(* CODESYS project DCCM_PCL_2.project
   Author: jrfsc
   Version: 0.0.0.0
   Title: DCCM_PCL_2

Project tree, tasks and I/O mapping:
  DCCM_PCL_2 : TM251MESC, Schneider Electric, order no. TM251MESC, version 5.1.9.35
      settings: OPCUA enable = False
    application Application
      libraries: IecRtsServices, 1.0.4.0 (Schneider Electric)
      task MAST (cyclic, interval 20 ms, priority 15, watchdog 100 ms x 1) calls INPUT_MAPPING, ROOM_1, ROOM_2, ROOM_3, ROOM_4, OUTPUT_MAPPING, SR_Main
      global variables GVL
      program SR_Main [FBD]
      program INPUT_MAPPING [ST]
      program OUTPUT_MAPPING [ST]
      FBs/
        function block DUTY [ST]
        function block DUTY_CHANGE [ST]
        function block FB_9StatesMonitoring [ST]
        function block FB_DUTY_DUTY_STANDBY_PUMP_SPD [ST]
        function block FB_FLOATING_VALVE [ST]
        function block FB_HEATING_OR_COOLING [ST]
        function block FB_OMODE [ST]
        function block FB_PMODE [ST]
        function block FB_SETPOINT_MODE [ST]
        function block FB_WATCHDOG [ST]
        function block LINEAR [ST]
        function block SATSP_CALC [ST]
        function block SB_HEATING_COOLING [ST]
        function block TERMINAL_LOAD [ST]
        program ISO_MODE [ST]
      Enumeration/
        data type ET_9STATE_MONITORING
        data type ET_OMODE
        data type ET_PMODE
      LIBRARY/
        function block FB_PULSE_GENERATOR [ST]
        function block FB_0_10V_TO_2_10V_OUTPUT [ST]
        function block FB_PCMS_WATCHDOG [ST]
      Library/
        function block FB_SETPOINT_RAMPING [ST]
      program ROOM_1 [FBD]
      program ROOM_4 [FBD]
      program ROOM_3 [FBD]
      program ROOM_2 [FBD]
      global variables DCCMNVL
      program SendDeprox [CFC]
      global variables PersistentVars
    IO_Bus : IO bus - TM3, Schneider Electric, version 5.1.9.35
      Module_1 : TM3AQ4/G, Schneider Electric, order no. TM3AQ4/G, version 1.0.0.16
          settings: KPI Configuration.KPI Configuration = 16; KPI Configuration.KPI Configuration = 16; KPI Configuration.KPI Configuration = 16; KPI Configuration.KPI Configuration = 16; KPI Configuration.KPI Configuration = 0; KPI Configuration.KPI Configuration = 0; KPI Configuration.KPI Configuration = 0; KPI Configuration.KPI Configuration = 0; KPI Configuration.KPI Configuration = 16; KPI Configuration.KPI Configuration = 39; KPI Configuration.KPI Configuration = 16; KPI Configuration.KPI Configuration = 39; KPI Configuration.KPI Configuration = 16; KPI Configuration.KPI Configuration = 39; KPI Configuration.KPI Configuration = 16; KPI Configuration.KPI Configuration = 39
          output qRM1_TRANSFER_DAMPER : INT  // QW0
          output qRM2_TRANSFER_DAMPER : INT  // QW1
          output qRM3_TRANSFER_DAMPER : INT  // QW2
          output qRM4_TRANSFER_DAMPER : INT  // QW3
          input  ibModule_1_IBStatusQW0 : BYTE  // IBStatusQW0
          input  ibModule_1_IBStatusQW1 : BYTE  // IBStatusQW1
          input  ibModule_1_IBStatusQW2 : BYTE  // IBStatusQW2
          input  ibModule_1_IBStatusQW3 : BYTE  // IBStatusQW3
      Module_2 : TM3AI8/G, Schneider Electric, order no. TM3AI8/G, version 1.0.0.27
          settings: KPI Configuration.KPI Configuration = 32; KPI Configuration.KPI Configuration = 32; KPI Configuration.KPI Configuration = 32; KPI Configuration.KPI Configuration = 32; KPI Configuration.KPI Configuration = 32; KPI Configuration.KPI Configuration = 32; KPI Configuration.KPI Configuration = 32; KPI Configuration.KPI Configuration = 32; KPI Configuration.KPI Configuration = 231; KPI Configuration.KPI Configuration = 255; KPI Configuration.KPI Configuration = 231; KPI Configuration.KPI Configuration = 255; KPI Configuration.KPI Configuration = 231; KPI Configuration.KPI Configuration = 255; KPI Configuration.KPI Configuration = 231; KPI Configuration.KPI Configuration = 255; KPI Configuration.KPI Configuration = 231; KPI Configuration.KPI Configuration = 255; KPI Configuration.KPI Configuration = 231; KPI Configuration.KPI Configuration = 255; KPI Configuration.KPI Configuration = 231; KPI Configuration.KPI Configuration = 255; KPI Configuration.KPI Configuration = 231; KPI Configuration.KPI Configuration = 255; KPI Configuration.KPI Configuration = 25; KPI Configuration.KPI Configuration = 0; KPI Configuration.KPI Configuration = 25; KPI Configuration.KPI Configuration = 0; KPI Configuration.KPI Configuration = 25; KPI Configuration.KPI Configuration = 0; KPI Configuration.KPI Configuration = 25; KPI Configuration.KPI Configuration = 0; KPI Configuration.KPI Configuration = 25; KPI Configuration.KPI Configuration = 0; KPI Configuration.KPI Configuration = 25; KPI Configuration.KPI Configuration = 0; KPI Configuration.KPI Configuration = 25; KPI Configuration.KPI Configuration = 0; KPI Configuration.KPI Configuration = 25; KPI Configuration.KPI Configuration = 0
          input  iRM1_DP_H_TO_R : INT  // IW0
          input  iRM1_DP_H_TO_A : INT  // IW1
          input  iRM1_DP_A_TO_R : INT  // IW2
          input  iRM2_DP_H_TO_R : INT  // IW3
          input  iRM2_DP_A_TO_R : INT  // IW4
          input  iRM2_3_DP_H_TO_A : INT  // IW5
          input  iRM3_DP_H_TO_R : INT  // IW6
          input  iRM3_DP_A_TO_R : INT  // IW7
          input  ibModule_2_IBStatusIW0 : BYTE  // IBStatusIW0
          input  ibModule_2_IBStatusIW1 : BYTE  // IBStatusIW1
          input  ibModule_2_IBStatusIW2 : BYTE  // IBStatusIW2
          input  ibModule_2_IBStatusIW3 : BYTE  // IBStatusIW3
          input  ibModule_2_IBStatusIW4 : BYTE  // IBStatusIW4
          input  ibModule_2_IBStatusIW5 : BYTE  // IBStatusIW5
          input  ibModule_2_IBStatusIW6 : BYTE  // IBStatusIW6
          input  ibModule_2_IBStatusIW7 : BYTE  // IBStatusIW7
      Module_3 : TM3AM6/G, Schneider Electric, order no. TM3AM6/G, version 1.0.0.23
          settings: KPI Configuration.KPI Configuration = 32; KPI Configuration.KPI Configuration = 32; KPI Configuration.KPI Configuration = 32; KPI Configuration.KPI Configuration = 32; KPI Configuration.KPI Configuration = 231; KPI Configuration.KPI Configuration = 255; KPI Configuration.KPI Configuration = 231; KPI Configuration.KPI Configuration = 255; KPI Configuration.KPI Configuration = 231; KPI Configuration.KPI Configuration = 255; KPI Configuration.KPI Configuration = 0; KPI Configuration.KPI Configuration = 25; KPI Configuration.KPI Configuration = 0; KPI Configuration.KPI Configuration = 25; KPI Configuration.KPI Configuration = 0; KPI Configuration.KPI Configuration = 25; KPI Configuration.KPI Configuration = 0; KPI Configuration.KPI Configuration = 100; KPI Configuration.KPI Configuration = 0
          input  iRM4_DP_H_TO_R : INT  // IW0
          input  iRM4_DP_H_TO_A : INT  // IW1
          input  iRM4_DP_A_TO_R : INT  // IW2
          input  iRM1_TRANSFER_DAMPER_FB : INT  // IW3
          input  ibModule_3_IBStatusIW0 : BYTE  // IBStatusIW0
          input  ibModule_3_IBStatusIW1 : BYTE  // IBStatusIW1
          input  ibModule_3_IBStatusIW2 : BYTE  // IBStatusIW2
          input  ibModule_3_IBStatusIW3 : BYTE  // IBStatusIW3
          input  ibModule_3_IBStatusQW0 : BYTE  // IBStatusQW0
          input  ibModule_3_IBStatusQW1 : BYTE  // IBStatusQW1
          unmapped channels: QW0, QW1
      Module_4 : TM3AM6/G, Schneider Electric, order no. TM3AM6/G, version 1.0.0.23
          settings: KPI Configuration.KPI Configuration = 32; KPI Configuration.KPI Configuration = 32; KPI Configuration.KPI Configuration = 32; KPI Configuration.KPI Configuration = 0; KPI Configuration.KPI Configuration = 0; KPI Configuration.KPI Configuration = 0; KPI Configuration.KPI Configuration = 100; KPI Configuration.KPI Configuration = 0; KPI Configuration.KPI Configuration = 100; KPI Configuration.KPI Configuration = 0; KPI Configuration.KPI Configuration = 100; KPI Configuration.KPI Configuration = 0
          input  iRM2_TRANSFER_DAMPER_FB : INT  // IW0
          input  iRM3_TRANSFER_DAMPER_FB : INT  // IW1
          input  iRM4_TRANSFER_DAMPER_FB : INT  // IW2
          input  ibModule_4_IBStatusIW0 : BYTE  // IBStatusIW0
          input  ibModule_4_IBStatusIW1 : BYTE  // IBStatusIW1
          input  ibModule_4_IBStatusIW2 : BYTE  // IBStatusIW2
          input  ibModule_4_IBStatusIW3 : BYTE  // IBStatusIW3
          input  ibModule_4_IBStatusQW0 : BYTE  // IBStatusQW0
          input  ibModule_4_IBStatusQW1 : BYTE  // IBStatusQW1
          unmapped channels: IW3, QW0, QW1
      Module_5 : TM3DM24R/G, Schneider Electric, order no. TM3DM24R/G, version 1.0.2.0
          input  iRM1_SUPPLY_DAMPER_STS : BOOL  // IW0.I0
          input  iRM2_SUPPLY_DAMPER_STS : BOOL  // IW0.I1
          input  iRM3_SUPPLY_DAMPER_STS : BOOL  // IW0.I2
          input  iRM4_SUPPLY_DAMPER_STS : BOOL  // IW0.I3
          input  iRM1_EXHAUST_DAMPER_STS : BOOL  // IW0.I4
          input  iRM2_EXHAUST_DAMPER_STS : BOOL  // IW0.I5
          input  iRM3_EXHAUST_DAMPER_STS : BOOL  // IW0.I6
          input  iRM4_EXHAUST_DAMPER_STS : BOOL  // IW0.I7
          input  iRM1_ISOLATION_MODE_SW : BOOL  // IW0.I8
          input  iRM1_DEPROX_MODE_SW : BOOL  // IW0.I9
          input  iRM1_ALARM_MUTE : BOOL  // IW0.I10
          input  iRM2_ISOLATION_MODE_SW : BOOL  // IW0.I11
          input  iRM2_DEPROX_MODE_SW : BOOL  // IW0.I12
          input  iRM2_ALARM_MUTE : BOOL  // IW0.I13
          input  iRM3_ISOLATION_MODE_SW : BOOL  // IW0.I14
          input  iRM3_DEPROX_MODE_SW : BOOL  // IW0.I15
          output qRM1_SUPPLY_DAMPER : BOOL  // QB0.Q0
          output qRM2_SUPPLY_DAMPER : BOOL  // QB0.Q1
          output qRM3_SUPPLY_DAMPER : BOOL  // QB0.Q2
          output qRM4_SUPPLY_DAMPER : BOOL  // QB0.Q3
          output qRM1_EXHAUST_DAMPER : BOOL  // QB0.Q4
          output qRM2_EXHAUST_DAMPER : BOOL  // QB0.Q5
          output qRM3_EXHAUST_DAMPER : BOOL  // QB0.Q6
          output qRM4_EXHAUST_DAMPER : BOOL  // QB0.Q7
          unmapped channels: IW0, QB0
      Module_6 : TM3DM24R/G, Schneider Electric, order no. TM3DM24R/G, version 1.0.2.0
          input  iRM3_ALARM_MUTE : BOOL  // IW0.I0
          input  iRM4_ISOLATION_MODE_SW : BOOL  // IW0.I1
          input  iRM4_DEPROX_MODE_SW : BOOL  // IW0.I2
          input  iRM4_ALARM_MUTE : BOOL  // IW0.I3
          output qRM1_NEGATIVE_LED : BOOL  // QB0.Q0
          output qRM1_DEPROX_LED : BOOL  // QB0.Q1
          output qRM1_ALARM_LED : BOOL  // QB0.Q2
          output qRM1_STANDBY_LED : BOOL  // QB0.Q3
          output qRM2_NEGATIVE_LED : BOOL  // QB0.Q4
          output qRM2_DEPROX_LED : BOOL  // QB0.Q5
          output qRM2_ALARM_LED : BOOL  // QB0.Q6
          output qRM2_STANDBY_LED : BOOL  // QB0.Q7
          unmapped channels: IW0, QB0
      Module_7 : TM3DQ16R/G, Schneider Electric, order no. TM3DQ16R/G, version 1.0.1.14
          output qRM3_NEGATIVE_LED : BOOL  // QW0.Q0
          output qRM3_DEPROX_LED : BOOL  // QW0.Q1
          output qRM3_ALARM_LED : BOOL  // QW0.Q2
          output qRM3_STANDBY_LED : BOOL  // QW0.Q3
          output qRM4_NEGATIVE_LED : BOOL  // QW0.Q4
          output qRM4_DEPROX_LED : BOOL  // QW0.Q5
          output qRM4_ALARM_LED : BOOL  // QW0.Q6
          output qRM4_STANDBY_LED : BOOL  // QW0.Q7
          output qRM1_BUZZER : BOOL  // QW0.Q8
          output qRM2_BUZZER : BOOL  // QW0.Q9
          output qRM3_BUZZER : BOOL  // QW0.Q10
          output qRM4_BUZZER : BOOL  // QW0.Q11
          unmapped channels: QW0
    COM_Bus : COM bus, Schneider Electric, version 5.1.9.35
    Ethernet_1 : Ethernet Network, Schneider Electric, version 5.1.9.35
        settings: WebServer = TRUE; FTP Server = FALSE; SoMachine Protocol = TRUE; Modbus Server = TRUE; NetManage Protocol = TRUE; SNMP protocol = FALSE; WebVisu protocol = FALSE; Secured Web Server = TRUE
    Serial_Line_1 : Serial line, Schneider Electric, version 5.1.9.35
      Machine_Expert_Network_Manager : Machine Expert-Network Manager, Schneider Electric, version 4.0.0.4
    CAN_1 : CANopen bus, Schneider Electric, version 5.1.9.35
*)

// DCCM_PCL_2/Application/Enumeration/ET_9STATE_MONITORING
{attribute 'qualified_only' := ''}
{attribute 'strict' := ''}
TYPE ET_9STATE_MONITORING :
(
	STOPPED := 0,
	RUNNING := 1,
	STARTING := 2,
	STOPPING := 3,
	START_FAIL := 4,
	STOP_FAIL := 5,
	UNEXPECTED_START := 6,
	UNEXPECTED_STOP := 7,
	FIRE_STOP := 8,
	UNKNOWN := 9
);
END_TYPE

// DCCM_PCL_2/Application/Enumeration/ET_OMODE
{attribute 'qualified_only' := ''}
{attribute 'strict' := ''}
TYPE ET_OMODE :
(
	UNOCC := 0,
	OPTSTART := 1,
	SCH := 2,
	AHRS := 3,
	MOTDETECT := 4,
	SETBACK := 7
);
END_TYPE

// DCCM_PCL_2/Application/Enumeration/ET_PMODE
{attribute 'qualified_only' := ''}
{attribute 'strict' := ''}
TYPE ET_PMODE :
(
	OFF_NORMAL := 0,
	OFF_PCMS := 1,
	OFF_Fire := 2,
	OFF_DMPRLOCK := 3,
	OFF_RESET := 4,
	Startup := 5,
	Purge := 6,
	RUN_NORMAL := 7
);
END_TYPE

// DCCM_PCL_2/Application/GVL
{attribute 'qualified_only'}
VAR_GLOBAL
	RM1_TRANSFER_DAMPER AT %MD500: REAL;
	RM2_TRANSFER_DAMPER AT %MD501: REAL;
	RM3_TRANSFER_DAMPER AT %MD502: REAL;
	RM4_TRANSFER_DAMPER AT %MD503: REAL;
	RM1_DP_H_TO_R AT %MD504: REAL;
	RM1_DP_H_TO_A AT %MD505: REAL;
	RM1_DP_A_TO_R AT %MD506: REAL;
	RM2_DP_H_TO_R AT %MD507: REAL;
	RM2_DP_A_TO_R AT %MD508: REAL;
	RM2_3_DP_H_TO_A AT %MD509: REAL;
	RM3_DP_H_TO_R AT %MD510: REAL;
	RM3_DP_A_TO_R AT %MD511: REAL;
	RM4_DP_H_TO_R AT %MD512: REAL;
	RM4_DP_H_TO_A AT %MD513: REAL;
	RM4_DP_A_TO_R AT %MD514: REAL;
	RM1_TRANSFER_DAMPER_FB AT %MD515: REAL;
	RM2_TRANSFER_DAMPER_FB AT %MD516: REAL;
	RM3_TRANSFER_DAMPER_FB AT %MD517: REAL;
	RM4_TRANSFER_DAMPER_FB AT %MD518: REAL;
	RM1_SUPPLY_DAMPER_STS AT %MX0.0: BOOL;
	RM2_SUPPLY_DAMPER_STS AT %MX0.1: BOOL;
	RM3_SUPPLY_DAMPER_STS AT %MX0.2: BOOL;
	RM4_SUPPLY_DAMPER_STS AT %MX0.3: BOOL;
	RM1_EXHAUST_DAMPER_STS AT %MX0.4: BOOL;
	RM2_EXHAUST_DAMPER_STS AT %MX0.5: BOOL;
	RM3_EXHAUST_DAMPER_STS AT %MX0.6: BOOL;
	RM4_EXHAUST_DAMPER_STS AT %MX0.7: BOOL;
	RM1_ISOLATION_MODE_SW AT %MX1.0: BOOL;
	RM1_DEPROX_MODE_SW AT %MX1.1: BOOL;
	RM1_ALARM_MUTE_SW AT %MX1.2: BOOL;
	RM2_ISOLATION_MODE_SW AT %MX1.3: BOOL;
	RM2_DEPROX_MODE_SW AT %MX1.4: BOOL;
	RM2_ALARM_MUTE_SW AT %MX1.5: BOOL;
	RM3_ISOLATION_MODE_SW AT %MX1.6: BOOL;
	RM3_DEPROX_MODE_SW AT %MX1.7: BOOL;
	RM1_SUPPLY_DAMPER AT %MX2.0: BOOL;
	RM2_SUPPLY_DAMPER AT %MX2.1: BOOL;
	RM3_SUPPLY_DAMPER AT %MX2.2: BOOL;
	RM4_SUPPLY_DAMPER AT %MX2.3: BOOL;
	RM1_EXHAUST_DAMPER AT %MX2.4: BOOL;
	RM2_EXHAUST_DAMPER AT %MX2.5: BOOL;
	RM3_EXHAUST_DAMPER AT %MX2.6: BOOL;
	RM4_EXHAUST_DAMPER AT %MX2.7: BOOL;
	RM3_ALARM_MUTE AT %MX3.0: BOOL;
	RM4_ISOLATION_MODE_SW AT %MX3.1: BOOL;
	RM4_DEPROX_MODE_SW AT %MX3.2: BOOL;
	RM4_ALARM_MUTE AT %MX3.3: BOOL;
	RM1_NEGATIVE_LED AT %MX3.4: BOOL;
	RM1_DEPROX_LED AT %MX3.5: BOOL;
	RM1_ALARM_LED AT %MX3.6: BOOL;
	RM1_STANDBY_LED AT %MX3.7: BOOL;
	RM2_NEGATIVE_LED AT %MX4.0: BOOL;
	RM2_DEPROX_LED AT %MX4.1: BOOL;
	RM2_ALARM_LED AT %MX4.2: BOOL;
	RM2_STANDBY_LED AT %MX4.3: BOOL;
	RM3_NEGATIVE_LED AT %MX4.4: BOOL;
	RM3_DEPROX_LED AT %MX4.5: BOOL;
	RM3_ALARM_LED AT %MX4.6: BOOL;
	RM3_STANDBY_LED AT %MX4.7: BOOL;
	RM4_NEGATIVE_LED AT %MX5.0: BOOL;
	RM4_ALARM_LED AT %MX5.1: BOOL;
	RM4_STANDBY_LED AT %MX5.2: BOOL;
	RM4_DEPROX_LED AT %MX5.3: BOOL;
	RM1_BUZZER AT %MX5.4: BOOL;
	RM2_BUZZER AT %MX5.5: BOOL;
	RM3_BUZZER AT %MX5.6: BOOL;
	RM4_BUZZER AT %MX5.7: BOOL;
	RM1_ISO_MODE AT %MW9000: INT;
	RM2_ISO_MODE AT %MW9001: INT;
	RM3_ISO_MODE AT %MW9002: INT;
	RM4_ISO_MODE AT %MW9003: INT;
	RM1_TRANSFER_DAMPER_MAN AT %MD523: REAL;
END_VAR
VAR_GLOBAL RETAIN PERSISTENT
	RM1_TRANSFER_DAMPER_MD AT %MX6.0: BOOL := TRUE;
END_VAR
VAR_GLOBAL
	RM2_TRANSFER_DAMPER_MAN AT %MD524: REAL;
END_VAR
VAR_GLOBAL RETAIN PERSISTENT
	RM2_TRANSFER_DAMPER_MD AT %MX6.1: BOOL := TRUE;
END_VAR
VAR_GLOBAL
	RM3_TRANSFER_DAMPER_MAN AT %MD525: REAL;
END_VAR
VAR_GLOBAL RETAIN PERSISTENT
	RM3_TRANSFER_DAMPER_MD AT %MX6.2: BOOL := TRUE;
END_VAR
VAR_GLOBAL
	RM4_TRANSFER_DAMPER_MAN AT %MD526: REAL;
END_VAR
VAR_GLOBAL RETAIN PERSISTENT
	RM4_TRANSFER_DAMPER_MD AT %MX6.3: BOOL := TRUE;
	RM1_DP1_SP AT %MD527: REAL := 8;
	RM2_DP1_SP AT %MD528: REAL := 8;
	RM3_DP1_SP AT %MD529: REAL := 8;
	RM4_DP1_SP AT %MD530: REAL := 8;
END_VAR
VAR_GLOBAL
	RM1_DP_ALM AT %MX6.4: BOOL;
	RM2_DP_ALM AT %MX6.5: BOOL;
	RM3_DP_ALM AT %MX6.6: BOOL;
	RM4_DP_ALM AT %MX6.7: BOOL;
	RM1_SUPPLY_DAMPER_MAN AT %MX7.0: BOOL;
END_VAR
VAR_GLOBAL RETAIN PERSISTENT
	RM1_SUPPLY_DAMPER_MD AT %MX7.1: BOOL := TRUE;
END_VAR
VAR_GLOBAL
	RM1_EXHAUST_DAMPER_MAN AT %MX7.2: BOOL;
END_VAR
VAR_GLOBAL RETAIN PERSISTENT
	RM1_EXHAUST_DAMPER_MD AT %MX7.3: BOOL := TRUE;
END_VAR
VAR_GLOBAL
	RM2_SUPPLY_DAMPER_MAN AT %MX7.4: BOOL;
END_VAR
VAR_GLOBAL RETAIN PERSISTENT
	RM2_SUPPLY_DAMPER_MD AT %MX7.5: BOOL := TRUE;
END_VAR
VAR_GLOBAL
	RM2_EXHAUST_DAMPER_MAN AT %MX7.6: BOOL;
END_VAR
VAR_GLOBAL RETAIN PERSISTENT
	RM2_EXHAUST_DAMPER_MD AT %MX7.7: BOOL := TRUE;
END_VAR
VAR_GLOBAL
	RM3_SUPPLY_DAMPER_MAN AT %MX8.0: BOOL;
END_VAR
VAR_GLOBAL RETAIN PERSISTENT
	RM3_SUPPLY_DAMPER_MD AT %MX8.1: BOOL := TRUE;
END_VAR
VAR_GLOBAL
	RM3_EXHAUST_DAMPER_MAN AT %MX8.2: BOOL;
END_VAR
VAR_GLOBAL RETAIN PERSISTENT
	RM3_EXHAUST_DAMPER_MD AT %MX8.3: BOOL := TRUE;
END_VAR
VAR_GLOBAL
	RM4_SUPPLY_DAMPER_MAN AT %MX8.4: BOOL;
END_VAR
VAR_GLOBAL RETAIN PERSISTENT
	RM4_SUPPLY_DAMPER_MD AT %MX8.5: BOOL := TRUE;
END_VAR
VAR_GLOBAL
	RM4_EXHAUST_DAMPER_MAN AT %MX8.6: BOOL;
END_VAR
VAR_GLOBAL RETAIN PERSISTENT
	RM4_EXHAUST_DAMPER_MD AT %MX8.7: BOOL := TRUE;
END_VAR
VAR_GLOBAL
	RM1_NEGATIVE_LED_MAN: BOOL;
	RM1_NEGATIVE_LED_MD: BOOL := TRUE;
	RM1_DEPROX_LED_MAN: BOOL;
	RM1_DEPROX_LED_MD: BOOL := TRUE;
	RM1_ALARM_LED_MAN: BOOL;
	RM1_ALARM_LED_MD: BOOL := TRUE;
	RM1_STANDBY_LED_MAN: BOOL;
	RM1_STANDBY_LED_MD: BOOL := TRUE;
	RM2_NEGATIVE_LED_MAN: BOOL;
	RM2_NEGATIVE_LED_MD: BOOL := TRUE;
	RM2_DEPROX_LED_MAN: BOOL;
	RM2_DEPROX_LED_MD: BOOL := TRUE;
	RM2_STANDBY_LED_MAN: BOOL;
	RM2_STANDBY_LED_MD: BOOL := TRUE;
	RM2_ALARM_LED_MAN: BOOL;
	RM2_ALARM_LED_MD: BOOL := TRUE;
	RM3_NEGATIVE_LED_MAN: BOOL;
	RM3_NEGATIVE_LED_MD: BOOL := TRUE;
	RM3_DEPROX_LED_MAN: BOOL;
	RM3_DEPROX_LED_MD: BOOL := TRUE;
	RM3_ALARM_LED_MAN: BOOL;
	RM3_ALARM_LED_MD: BOOL := TRUE;
	RM3_STANDBY_LED_MAN: BOOL;
	RM3_STANDBY_LED_MD: BOOL := TRUE;
	RM4_NEGATIVE_LED_MAN: BOOL;
	RM4_NEGATIVE_LED_MD: BOOL := TRUE;
	RM4_DEPROX_LED_MAN: BOOL;
	RM4_DEPROX_LED_MD: BOOL := TRUE;
	RM4_ALARM_LED_MAN: BOOL;
	RM4_ALARM_LED_MD: BOOL := TRUE;
	RM4_STANDBY_LED_MAN: BOOL;
	RM4_STANDBY_LED_MD: BOOL := TRUE;
END_VAR
VAR_GLOBAL RETAIN PERSISTENT
	RM1_TRANSFER_DAMPER_ISO_SP AT %MD535: REAL := 15;
	RM2_TRANSFER_DAMPER_ISO_SP AT %MD536: REAL := 15;
	RM3_TRANSFER_DAMPER_ISO_SP AT %MD537: REAL := 15;
	RM4_TRANSFER_DAMPER_ISO_SP AT %MD538: REAL := 10;
END_VAR
VAR_GLOBAL
	RM1_BUZZER_MAN: BOOL;
	RM1_BUZZER_MD: BOOL := TRUE;
	RM2_BUZZER_MAN: BOOL;
	RM2_BUZZER_MD: BOOL := TRUE;
	RM3_BUZZER_MAN: BOOL;
	RM3_BUZZER_MD: BOOL := TRUE;
	RM4_BUZZER_MAN: BOOL;
	RM4_BUZZER_MD: BOOL := TRUE;
END_VAR
VAR_GLOBAL RETAIN PERSISTENT
	RM1_ALARM_DELAY AT %MD539: real := 180;
	RM2_ALARM_DELAY AT %MD540: real := 180;
	RM3_ALARM_DELAY AT %MD541: real := 180;
	RM4_ALARM_DELAY AT %MD542: real := 180;
END_VAR
VAR_GLOBAL
	DEPROX_TOTAL AT %MW9004: INT;
END_VAR
VAR_GLOBAL RETAIN PERSISTENT
	RM1_DP2_SP AT %MD543: REAL;
	RM1_DP3_SP AT %MD544: REAL;
	RM2_DP2_SP AT %MD545: REAL;
	RM2_DP3_SP AT %MD546: REAL;
	RM3_DP2_SP AT %MD547: REAL;
	RM3_DP3_SP AT %MD548: REAL;
	RM4_DP2_SP AT %MD549: REAL;
	RM4_DP3_SP AT %MD550: REAL;
	RM1_TRANSFER_DAMPER_DEP_SP AT %MD551: REAL;
	RM2_TRANSFER_DAMPER_DEP_SP AT %MD552: REAL;
	RM3_TRANSFER_DAMPER_DEP_SP AT %MD553: REAL;
	RM4_TRANSFER_DAMPER_DEP_SP AT %MD554: REAL;
END_VAR

// DCCM_PCL_2/Application/DCCMNVL
{attribute 'qualified_only'}
VAR_GLOBAL
	RM1_ISO_MODE AT %MW9000: INT;
	RM2_ISO_MODE AT %MW9001: INT;
	RM3_ISO_MODE AT %MW9002: INT;
	RM4_ISO_MODE AT %MW9003: INT;
END_VAR

// DCCM_PCL_2/Application/PersistentVars
{attribute 'qualified_only'}
VAR_GLOBAL PERSISTENT RETAIN
	// Generated instance path of persistent variable
	GVL.RM1_TRANSFER_DAMPER_MD: BOOL := TRUE;
	// Generated instance path of persistent variable
	GVL.RM2_TRANSFER_DAMPER_MD: BOOL := TRUE;
	// Generated instance path of persistent variable
	GVL.RM3_TRANSFER_DAMPER_MD: BOOL := TRUE;
	// Generated instance path of persistent variable
	GVL.RM4_TRANSFER_DAMPER_MD: BOOL := TRUE;
	// Generated instance path of persistent variable
	GVL.RM1_DP1_SP: REAL := -5;
	// Generated instance path of persistent variable
	GVL.RM2_DP1_SP: REAL := -5;
	// Generated instance path of persistent variable
	GVL.RM3_DP1_SP: REAL := -5;
	// Generated instance path of persistent variable
	GVL.RM4_DP1_SP: REAL := -5;
	// Generated instance path of persistent variable
	GVL.RM1_SUPPLY_DAMPER_MD: BOOL := TRUE;
	// Generated instance path of persistent variable
	GVL.RM1_EXHAUST_DAMPER_MD: BOOL := TRUE;
	// Generated instance path of persistent variable
	GVL.RM2_SUPPLY_DAMPER_MD: BOOL := TRUE;
	// Generated instance path of persistent variable
	GVL.RM2_EXHAUST_DAMPER_MD: BOOL := TRUE;
	// Generated instance path of persistent variable
	GVL.RM3_SUPPLY_DAMPER_MD: BOOL := TRUE;
	// Generated instance path of persistent variable
	GVL.RM3_EXHAUST_DAMPER_MD: BOOL := TRUE;
	// Generated instance path of persistent variable
	GVL.RM4_SUPPLY_DAMPER_MD: BOOL := TRUE;
	// Generated instance path of persistent variable
	GVL.RM4_EXHAUST_DAMPER_MD: BOOL := TRUE;
	// Generated instance path of persistent variable
	GVL.RM1_TRANSFER_DAMPER_ISO_SP: REAL := 15.0;
	// Generated instance path of persistent variable
	GVL.RM2_TRANSFER_DAMPER_ISO_SP: REAL := 15.0;
	// Generated instance path of persistent variable
	GVL.RM3_TRANSFER_DAMPER_ISO_SP: REAL := 15.0;
	// Generated instance path of persistent variable
	GVL.RM4_TRANSFER_DAMPER_ISO_SP: REAL := 10.0;
	// Generated instance path of persistent variable
	GVL.RM1_ALARM_DELAY: REAL := 180.0;
	// Generated instance path of persistent variable
	GVL.RM2_ALARM_DELAY: REAL := 180.0;
	// Generated instance path of persistent variable
	GVL.RM3_ALARM_DELAY: REAL := 180.0;
	// Generated instance path of persistent variable
	GVL.RM4_ALARM_DELAY: REAL := 180.0;
	// Generated instance path of persistent variable
	GVL.RM1_DP2_SP: REAL := -5;
	// Generated instance path of persistent variable
	GVL.RM1_DP3_SP: REAL := -5;
	// Generated instance path of persistent variable
	GVL.RM2_DP2_SP: REAL := -5;
	// Generated instance path of persistent variable
	GVL.RM2_DP3_SP: REAL := -5;
	// Generated instance path of persistent variable
	GVL.RM3_DP2_SP: REAL := -5;
	// Generated instance path of persistent variable
	GVL.RM3_DP3_SP: REAL := -5;
	// Generated instance path of persistent variable
	GVL.RM4_DP2_SP: REAL := -5;
	// Generated instance path of persistent variable
	GVL.RM4_DP3_SP: REAL := -5;
	// Generated instance path of persistent variable
	GVL.RM1_TRANSFER_DAMPER_DEP_SP: REAL;
	// Generated instance path of persistent variable
	GVL.RM2_TRANSFER_DAMPER_DEP_SP: REAL;
	// Generated instance path of persistent variable
	GVL.RM3_TRANSFER_DAMPER_DEP_SP: REAL;
	// Generated instance path of persistent variable
	GVL.RM4_TRANSFER_DAMPER_DEP_SP: REAL;
END_VAR

// DCCM_PCL_2/Application/INPUT_MAPPING
PROGRAM INPUT_MAPPING
VAR
		voltage_converter: FB_0_10V_TO_2_10V_OUTPUT;
END_VAR

//MAPPING HARDWARE INPUTS TO MEMORY WORDS

GVL.RM1_DP_H_TO_R := TO_REAL(iRM1_DP_H_TO_R);								//MODULE 2 TM3AI8 INPUT 0
GVL.RM1_DP_H_TO_A := TO_REAL(iRM1_DP_H_TO_A);								//MODULE 2 TM3AI8 INPUT 1
GVL.RM1_DP_A_TO_R := TO_REAL(iRM1_DP_A_TO_R);								//MODULE 2 TM3AI8 INPUT 2
GVL.RM2_DP_H_TO_R := TO_REAL(IRM2_DP_H_TO_R);								//MODULE 2 TM3AI8 INPUT 3
GVL.RM2_DP_A_TO_R := TO_REAL(iRM2_DP_A_TO_R);								//MODULE 2 TM3AI8 INPUT 4
GVL.RM2_3_DP_H_TO_A := TO_REAL(iRM2_3_DP_H_TO_A);							//MODULE 2 TM3AI8 INPUT 5
GVL.RM3_DP_H_TO_R := TO_REAL(iRM3_DP_H_TO_R);								//MODULE 2 TM3AI8 INPUT 6
GVL.RM3_DP_A_TO_R := TO_REAL(iRM3_DP_A_TO_R);								//MODULE 2 TM3AI8 INPUT 7

GVL.RM4_DP_H_TO_R := TO_REAL(iRM4_DP_H_TO_R);								//MODULE 3 TM3AM6 INPUT 0
GVL.RM4_DP_H_TO_A := TO_REAL(iRM4_DP_H_TO_A);								//MODULE 3 TM3AM6 INPUT 1
GVL.RM4_DP_A_TO_R := TO_REAL(iRM4_DP_A_TO_R);		
						//MODULE 3 TM3AM6 INPUT 2
//GVL.RM1_TRANSFER_DAMPER_FB := TO_REAL(iRM1_TRANSFER_DAMPER_FB);				//MODULE 3 TM3AM6 INPUT 3
//GVL.RM2_TRANSFER_DAMPER_FB := TO_REAL(iRM2_TRANSFER_DAMPER_FB);				//MODULE 4 TM3AM6 INPUT 0
//GVL.RM3_TRANSFER_DAMPER_FB := TO_REAL(iRM3_TRANSFER_DAMPER_FB);				//MODULE 4 TM3AM6 INPUT 1
//GVL.RM4_TRANSFER_DAMPER_FB := TO_REAL(iRM4_TRANSFER_DAMPER_FB);				//MODULE 4 TM3AM6 INPUT 2


GVL.RM1_TRANSFER_DAMPER_FB :=100-((((iRM1_TRANSFER_DAMPER_FB-100) * 100/80))+100);
GVL.RM2_TRANSFER_DAMPER_FB :=100-((((iRM2_TRANSFER_DAMPER_FB-100) * 100/80))+100);
GVL.RM3_TRANSFER_DAMPER_FB :=100-((((iRM3_TRANSFER_DAMPER_FB-100) * 100/80))+100);
GVL.RM4_TRANSFER_DAMPER_FB :=100-((((iRM4_TRANSFER_DAMPER_FB-100) * 100/80))+100);  //AI0  0v=open 10v=close



GVL.RM1_SUPPLY_DAMPER_STS := iRM1_SUPPLY_DAMPER_STS;						//MODULE 5 TM3DM24R INPUT 0
GVL.RM2_SUPPLY_DAMPER_STS := iRM2_SUPPLY_DAMPER_STS;						//MODULE 5 TM3DM24R INPUT 1
GVL.RM3_SUPPLY_DAMPER_STS := iRM3_SUPPLY_DAMPER_STS;						//MODULE 5 TM3DM24R INPUT 2
GVL.RM4_SUPPLY_DAMPER_STS := iRM4_SUPPLY_DAMPER_STS;						//MODULE 5 TM3DM24R INPUT 3
GVL.RM1_EXHAUST_DAMPER_STS := iRM1_EXHAUST_DAMPER_STS;						//MODULE 5 TM3DM24R INPUT 4
GVL.RM2_EXHAUST_DAMPER_STS := iRM2_EXHAUST_DAMPER_STS;						//MODULE 5 TM3DM24R INPUT 5
GVL.RM3_EXHAUST_DAMPER_STS := iRM3_EXHAUST_DAMPER_STS;						//MODULE 5 TM3DM24R INPUT 6
GVL.RM4_EXHAUST_DAMPER_STS := iRM4_EXHAUST_DAMPER_STS;						//MODULE 5 TM3DM24R INPUT 7
GVL.RM1_ISOLATION_MODE_SW := iRM1_ISOLATION_MODE_SW;						//MODULE 5 TM3DM24R INPUT 8
GVL.RM1_DEPROX_MODE_SW := iRM1_DEPROX_MODE_SW;								//MODULE 5 TM3DM24R INPUT 9
GVL.RM1_ALARM_MUTE_SW := iRM1_ALARM_MUTE;									//MODULE 5 TM3DM24R INPUT 10
GVL.RM2_ISOLATION_MODE_SW := iRM2_ISOLATION_MODE_SW;						//MODULE 5 TM3DM24R INPUT 11
GVL.RM2_DEPROX_MODE_SW := iRM2_DEPROX_MODE_SW;								//MODULE 5 TM3DM24R INPUT 12
GVL.RM2_ALARM_MUTE_SW := iRM2_ALARM_MUTE;									//MODULE 5 TM3DM24R INPUT 13
GVL.RM3_ISOLATION_MODE_SW := iRM3_ISOLATION_MODE_SW;						//MODULE 5 TM3DM24R INPUT 14
GVL.RM3_DEPROX_MODE_SW := iRM3_DEPROX_MODE_SW;								//MODULE 5 TM3DM24R INPUT 15

GVL.RM3_ALARM_MUTE := iRM3_ALARM_MUTE;										//MODULE 6 TM3DM24R INPUT 0
GVL.RM4_ISOLATION_MODE_SW := iRM4_ISOLATION_MODE_SW;						//MODULE 6 TM3DM24R INPUT 1
GVL.RM4_DEPROX_MODE_SW := iRM4_DEPROX_MODE_SW;								//MODULE 6 TM3DM24R INPUT 2
GVL.RM4_ALARM_MUTE := iRM4_ALARM_MUTE;										//MODULE 6 TM3DM24R INPUT 3

END_PROGRAM

// DCCM_PCL_2/Application/LIBRARY/FB_0_10V_TO_2_10V_OUTPUT
FUNCTION_BLOCK FB_0_10V_TO_2_10V_OUTPUT
VAR_OUTPUT
	// 0-10V = 0-100%
	OUT_PRCT: REAL;
END_VAR
VAR_INPUT
	// 2-10V = 0-100%
	IN_PRCT: REAL;
END_VAR

OUT_PRCT := ((IN_PRCT * 0.08) + 2) * 10;

END_FUNCTION_BLOCK

// DCCM_PCL_2/Application/ROOM_1
PROGRAM ROOM_1
VAR
	TON_0: TON;
	TOF_0: TOF;
	TOF_1: TOF;
	FLASHING: BOOL;
	FB_PULSE_GENERATOR_0: FB_PULSE_GENERATOR;
END_VAR
VAR // added by the converter: edge detectors and wires of the graphical bodies
    _rt1 : R_TRIG;
END_VAR

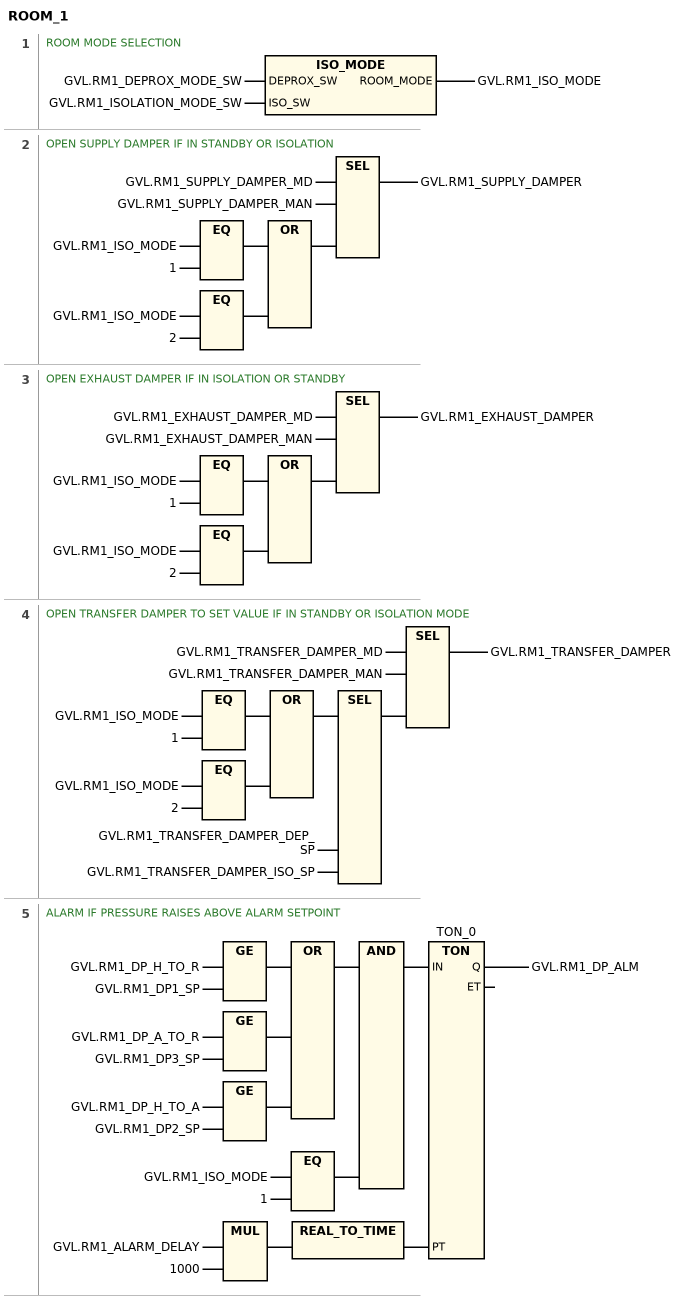
// NETWORK 1
// ROOM MODE SELECTION
ISO_MODE(DEPROX_SW := GVL.RM1_DEPROX_MODE_SW, ISO_SW := GVL.RM1_ISOLATION_MODE_SW);
GVL.RM1_ISO_MODE := ISO_MODE.ROOM_MODE;

// NETWORK 2
// OPEN SUPPLY DAMPER IF IN STANDBY OR ISOLATION
GVL.RM1_SUPPLY_DAMPER := SEL(GVL.RM1_SUPPLY_DAMPER_MD, GVL.RM1_SUPPLY_DAMPER_MAN, GVL.RM1_ISO_MODE = 1 OR GVL.RM1_ISO_MODE = 2);

// NETWORK 3
// OPEN EXHAUST DAMPER IF IN ISOLATION OR STANDBY
GVL.RM1_EXHAUST_DAMPER := SEL(GVL.RM1_EXHAUST_DAMPER_MD, GVL.RM1_EXHAUST_DAMPER_MAN, GVL.RM1_ISO_MODE = 1 OR GVL.RM1_ISO_MODE = 2);

// NETWORK 4
// OPEN TRANSFER DAMPER TO SET VALUE IF IN STANDBY OR ISOLATION MODE
GVL.RM1_TRANSFER_DAMPER := SEL(GVL.RM1_TRANSFER_DAMPER_MD, GVL.RM1_TRANSFER_DAMPER_MAN, SEL(GVL.RM1_ISO_MODE = 1 OR GVL.RM1_ISO_MODE = 2, GVL.RM1_TRANSFER_DAMPER_DEP_SP, GVL.RM1_TRANSFER_DAMPER_ISO_SP));

// NETWORK 5
// ALARM IF PRESSURE RAISES ABOVE ALARM SETPOINT
TON_0(IN := (GVL.RM1_DP_H_TO_R >= GVL.RM1_DP1_SP OR GVL.RM1_DP_A_TO_R >= GVL.RM1_DP3_SP OR GVL.RM1_DP_H_TO_A >= GVL.RM1_DP2_SP) AND GVL.RM1_ISO_MODE = 1, PT := REAL_TO_TIME(GVL.RM1_ALARM_DELAY * 1000)); // TON
GVL.RM1_DP_ALM := TON_0.Q;

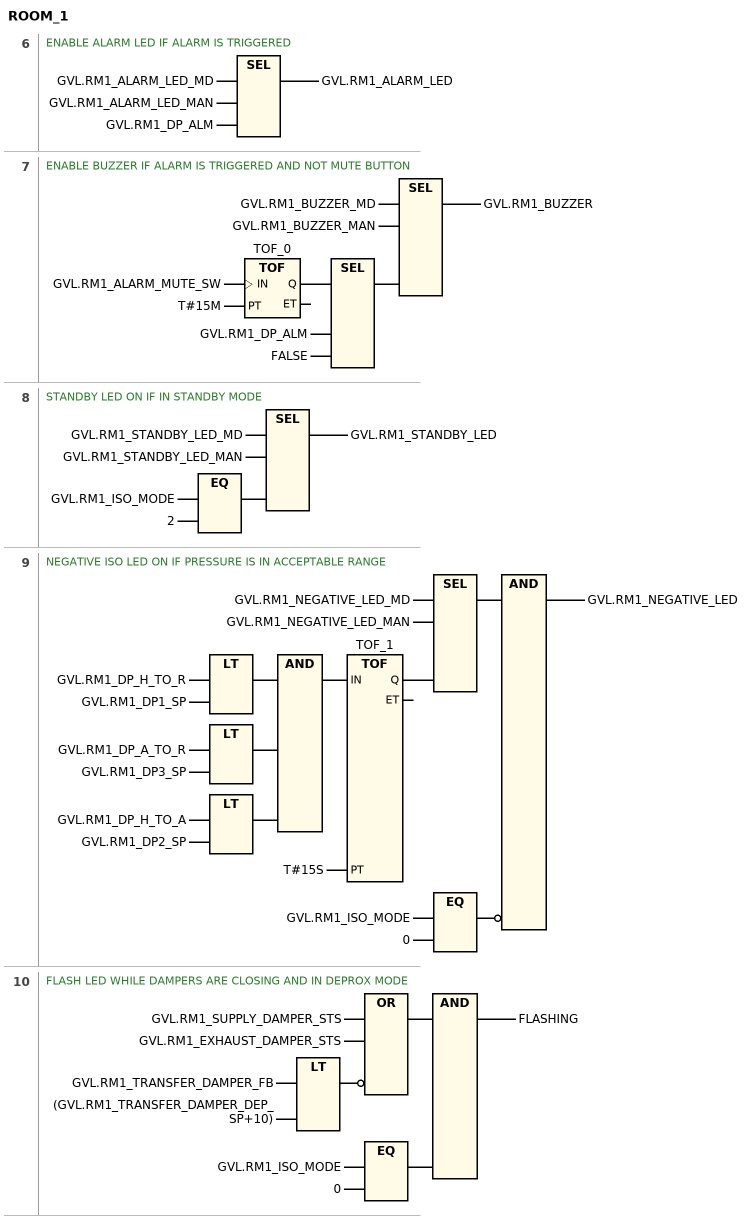
// NETWORK 6
// ENABLE ALARM LED IF ALARM IS TRIGGERED
GVL.RM1_ALARM_LED := SEL(GVL.RM1_ALARM_LED_MD, GVL.RM1_ALARM_LED_MAN, GVL.RM1_DP_ALM);

// NETWORK 7
// ENABLE BUZZER IF ALARM IS TRIGGERED AND NOT MUTE BUTTON
_rt1(CLK := GVL.RM1_ALARM_MUTE_SW);
TOF_0(IN := _rt1.Q, PT := T#15M); // TOF
GVL.RM1_BUZZER := SEL(GVL.RM1_BUZZER_MD, GVL.RM1_BUZZER_MAN, SEL(TOF_0.Q, GVL.RM1_DP_ALM, FALSE));

// NETWORK 8
// STANDBY LED ON IF IN STANDBY MODE
GVL.RM1_STANDBY_LED := SEL(GVL.RM1_STANDBY_LED_MD, GVL.RM1_STANDBY_LED_MAN, GVL.RM1_ISO_MODE = 2);

// NETWORK 9
// NEGATIVE ISO LED ON IF PRESSURE IS IN ACCEPTABLE RANGE
TOF_1(IN := GVL.RM1_DP_H_TO_R < GVL.RM1_DP1_SP AND GVL.RM1_DP_A_TO_R < GVL.RM1_DP3_SP AND GVL.RM1_DP_H_TO_A < GVL.RM1_DP2_SP, PT := T#15S); // TOF
GVL.RM1_NEGATIVE_LED := SEL(GVL.RM1_NEGATIVE_LED_MD, GVL.RM1_NEGATIVE_LED_MAN, TOF_1.Q) AND NOT (GVL.RM1_ISO_MODE = 0);

// NETWORK 10
// FLASH LED WHILE DAMPERS ARE CLOSING AND IN DEPROX MODE
FLASHING := (GVL.RM1_SUPPLY_DAMPER_STS OR GVL.RM1_EXHAUST_DAMPER_STS OR NOT (GVL.RM1_TRANSFER_DAMPER_FB < ((GVL.RM1_TRANSFER_DAMPER_DEP_SP+10)))) AND GVL.RM1_ISO_MODE = 0;

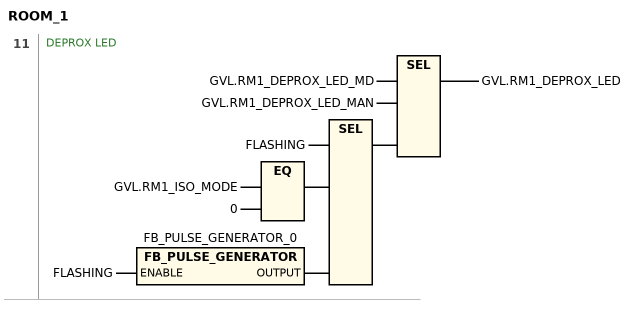
// NETWORK 11
// DEPROX LED
FB_PULSE_GENERATOR_0(ENABLE := FLASHING); // FB_PULSE_GENERATOR
GVL.RM1_DEPROX_LED := SEL(GVL.RM1_DEPROX_LED_MD, GVL.RM1_DEPROX_LED_MAN, SEL(FLASHING, GVL.RM1_ISO_MODE = 0, FB_PULSE_GENERATOR_0.OUTPUT));

END_PROGRAM

// DCCM_PCL_2/Application/FBs/ISO_MODE
PROGRAM ISO_MODE
VAR_INPUT
	DEPROX_SW: BOOL;
	ISO_SW: BOOL;
END_VAR
VAR_OUTPUT
	ROOM_MODE: INT;
END_VAR

(*
	ROOM MODE SWITCHING
	DEPROX = 0
	ISOLATION MODE = 1
	STANDBY = 2
	ERROR = 3
*)

IF (DEPROX_SW = TRUE AND ISO_SW = FALSE) THEN
	ROOM_MODE := 0;		//IF DEPROX SWITCH, THEN ENTER DEPROX MODE
ELSIF (ISO_SW = TRUE AND DEPROX_SW = FALSE) THEN
	ROOM_MODE := 1;		//IF ISO SWITCH, THEN ENTER ISOLATION MODE
ELSIF(ISO_SW = TRUE AND DEPROX_SW = TRUE) THEN
	ROOM_MODE := 3;		//IF BOTH SWITCHES, MODE IS IN ERROR
ELSE
	ROOM_MODE := 2;		//IF NEITHER SWITCH, ROOM IN STANDBY
END_IF;

END_PROGRAM

// DCCM_PCL_2/Application/LIBRARY/FB_PULSE_GENERATOR
FUNCTION_BLOCK FB_PULSE_GENERATOR
VAR_INPUT
	ENABLE: BOOL;
END_VAR
VAR_OUTPUT
	OUTPUT: BOOL;
END_VAR
VAR
	PULSESTATE: BOOL;
	PULSETIME: INT;
END_VAR


IF (ENABLE) THEN
	IF(PULSETIME > 100) THEN
		PULSESTATE := NOT PULSESTATE;
		PULSETIME := 0;
	END_IF;
	IF (PULSETIME < 0) THEN
		PULSETIME := 0;
	END_IF;
ELSE
	PULSESTATE := FALSE;
	PULSETIME := 0;
END_IF;

PULSETIME := PULSETIME +1;

OUTPUT := PULSESTATE;

END_FUNCTION_BLOCK

// DCCM_PCL_2/Application/ROOM_2
PROGRAM ROOM_2
VAR
	TON_0: TON;
	TOF_0: TOF;
	TOF_1: TOF;
	FLASHING: BOOL;
	FB_PULSE_GENERATOR_1: FB_PULSE_GENERATOR;
END_VAR
VAR // added by the converter: edge detectors and wires of the graphical bodies
    _rt1 : R_TRIG;
END_VAR

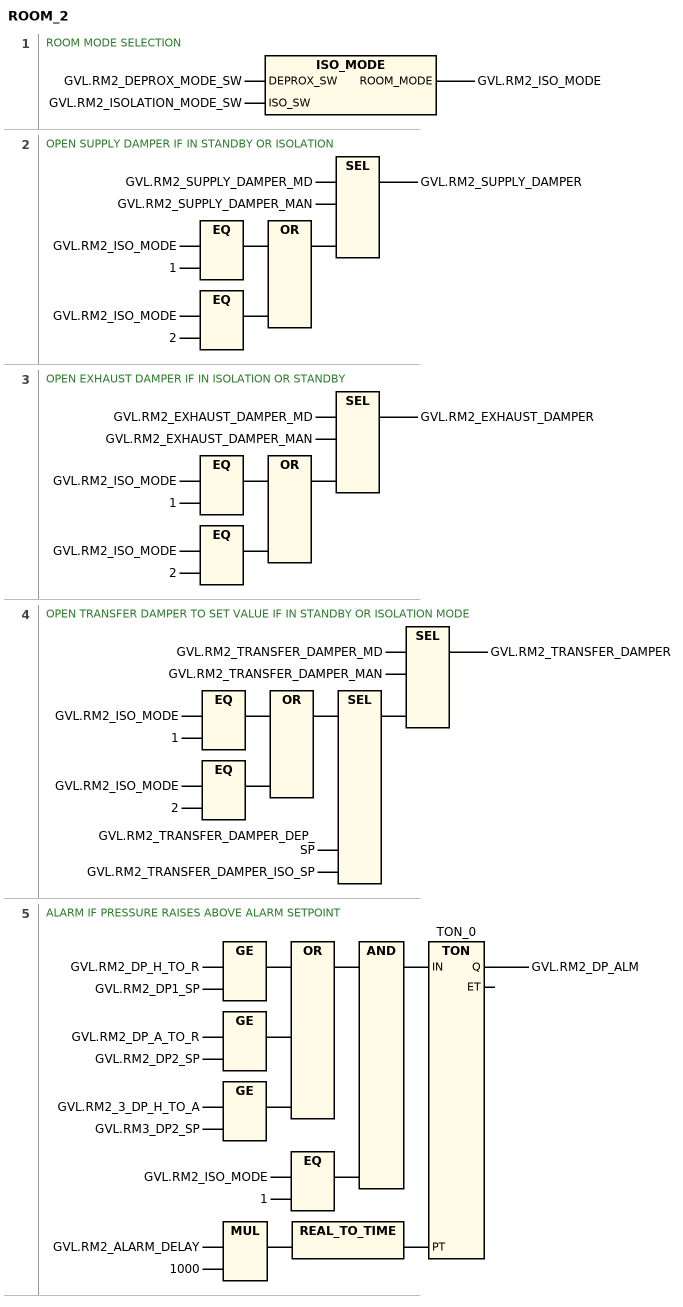
// NETWORK 1
// ROOM MODE SELECTION
ISO_MODE(DEPROX_SW := GVL.RM2_DEPROX_MODE_SW, ISO_SW := GVL.RM2_ISOLATION_MODE_SW);
GVL.RM2_ISO_MODE := ISO_MODE.ROOM_MODE;

// NETWORK 2
// OPEN SUPPLY DAMPER IF IN STANDBY OR ISOLATION
GVL.RM2_SUPPLY_DAMPER := SEL(GVL.RM2_SUPPLY_DAMPER_MD, GVL.RM2_SUPPLY_DAMPER_MAN, GVL.RM2_ISO_MODE = 1 OR GVL.RM2_ISO_MODE = 2);

// NETWORK 3
// OPEN EXHAUST DAMPER IF IN ISOLATION OR STANDBY
GVL.RM2_EXHAUST_DAMPER := SEL(GVL.RM2_EXHAUST_DAMPER_MD, GVL.RM2_EXHAUST_DAMPER_MAN, GVL.RM2_ISO_MODE = 1 OR GVL.RM2_ISO_MODE = 2);

// NETWORK 4
// OPEN TRANSFER DAMPER TO SET VALUE IF IN STANDBY OR ISOLATION MODE
GVL.RM2_TRANSFER_DAMPER := SEL(GVL.RM2_TRANSFER_DAMPER_MD, GVL.RM2_TRANSFER_DAMPER_MAN, SEL(GVL.RM2_ISO_MODE = 1 OR GVL.RM2_ISO_MODE = 2, GVL.RM2_TRANSFER_DAMPER_DEP_SP, GVL.RM2_TRANSFER_DAMPER_ISO_SP));

// NETWORK 5
// ALARM IF PRESSURE RAISES ABOVE ALARM SETPOINT
TON_0(IN := (GVL.RM2_DP_H_TO_R >= GVL.RM2_DP1_SP OR GVL.RM2_DP_A_TO_R >= GVL.RM2_DP2_SP OR GVL.RM2_3_DP_H_TO_A >= GVL.RM3_DP2_SP) AND GVL.RM2_ISO_MODE = 1, PT := REAL_TO_TIME(GVL.RM2_ALARM_DELAY * 1000)); // TON
GVL.RM2_DP_ALM := TON_0.Q;

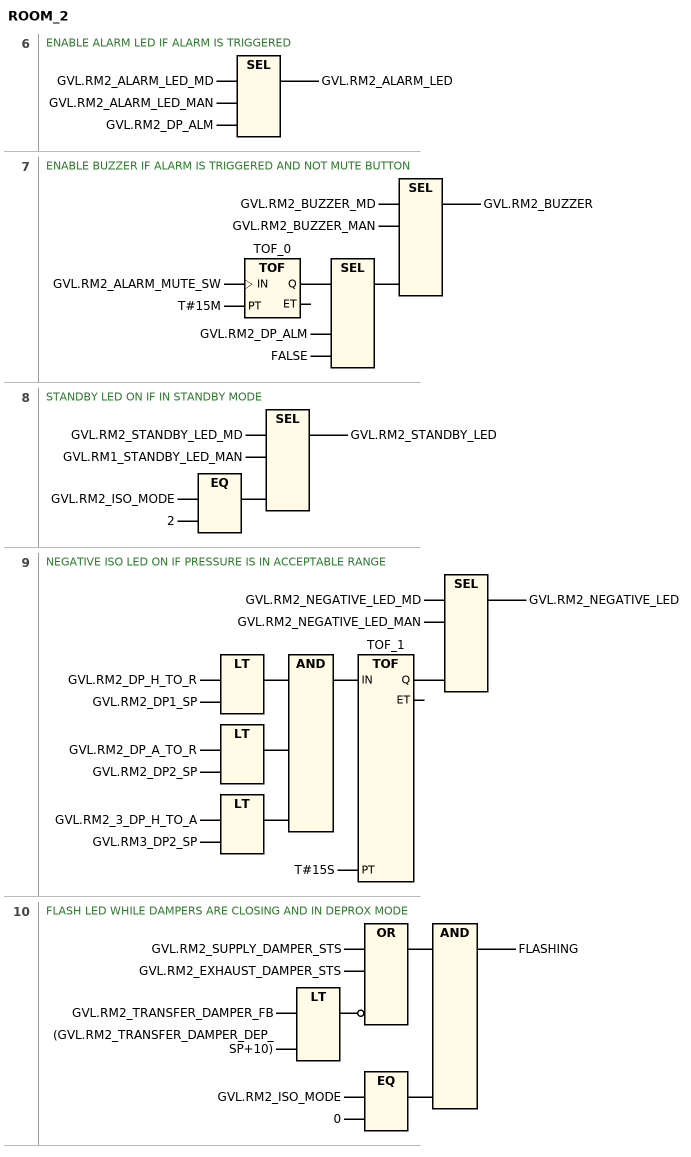
// NETWORK 6
// ENABLE ALARM LED IF ALARM IS TRIGGERED
GVL.RM2_ALARM_LED := SEL(GVL.RM2_ALARM_LED_MD, GVL.RM2_ALARM_LED_MAN, GVL.RM2_DP_ALM);

// NETWORK 7
// ENABLE BUZZER IF ALARM IS TRIGGERED AND NOT MUTE BUTTON
_rt1(CLK := GVL.RM2_ALARM_MUTE_SW);
TOF_0(IN := _rt1.Q, PT := T#15M); // TOF
GVL.RM2_BUZZER := SEL(GVL.RM2_BUZZER_MD, GVL.RM2_BUZZER_MAN, SEL(TOF_0.Q, GVL.RM2_DP_ALM, FALSE));

// NETWORK 8
// STANDBY LED ON IF IN STANDBY MODE
GVL.RM2_STANDBY_LED := SEL(GVL.RM2_STANDBY_LED_MD, GVL.RM1_STANDBY_LED_MAN, GVL.RM2_ISO_MODE = 2);

// NETWORK 9
// NEGATIVE ISO LED ON IF PRESSURE IS IN ACCEPTABLE RANGE
TOF_1(IN := GVL.RM2_DP_H_TO_R < GVL.RM2_DP1_SP AND GVL.RM2_DP_A_TO_R < GVL.RM2_DP2_SP AND GVL.RM2_3_DP_H_TO_A < GVL.RM3_DP2_SP, PT := T#15S); // TOF
GVL.RM2_NEGATIVE_LED := SEL(GVL.RM2_NEGATIVE_LED_MD, GVL.RM2_NEGATIVE_LED_MAN, TOF_1.Q);

// NETWORK 10
// FLASH LED WHILE DAMPERS ARE CLOSING AND IN DEPROX MODE
FLASHING := (GVL.RM2_SUPPLY_DAMPER_STS OR GVL.RM2_EXHAUST_DAMPER_STS OR NOT (GVL.RM2_TRANSFER_DAMPER_FB < ((GVL.RM2_TRANSFER_DAMPER_DEP_SP+10)))) AND GVL.RM2_ISO_MODE = 0;

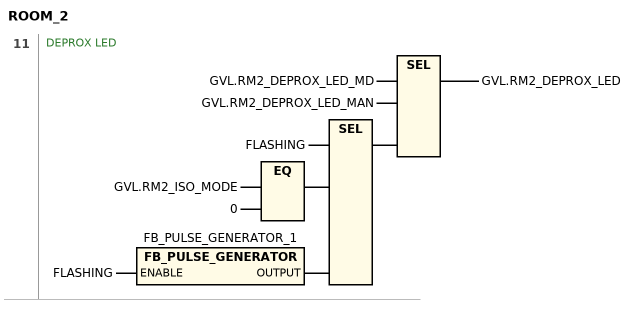
// NETWORK 11
// DEPROX LED
FB_PULSE_GENERATOR_1(ENABLE := FLASHING); // FB_PULSE_GENERATOR
GVL.RM2_DEPROX_LED := SEL(GVL.RM2_DEPROX_LED_MD, GVL.RM2_DEPROX_LED_MAN, SEL(FLASHING, GVL.RM2_ISO_MODE = 0, FB_PULSE_GENERATOR_1.OUTPUT));

END_PROGRAM

// DCCM_PCL_2/Application/ROOM_3
PROGRAM ROOM_3
VAR
	TON_0: TON;
	TOF_0: TOF;
	TOF_1: TOF;
	FLASHING: BOOL;
	FB_PULSE_GENERATOR_2: FB_PULSE_GENERATOR;
END_VAR
VAR // added by the converter: edge detectors and wires of the graphical bodies
    _rt1 : R_TRIG;
END_VAR

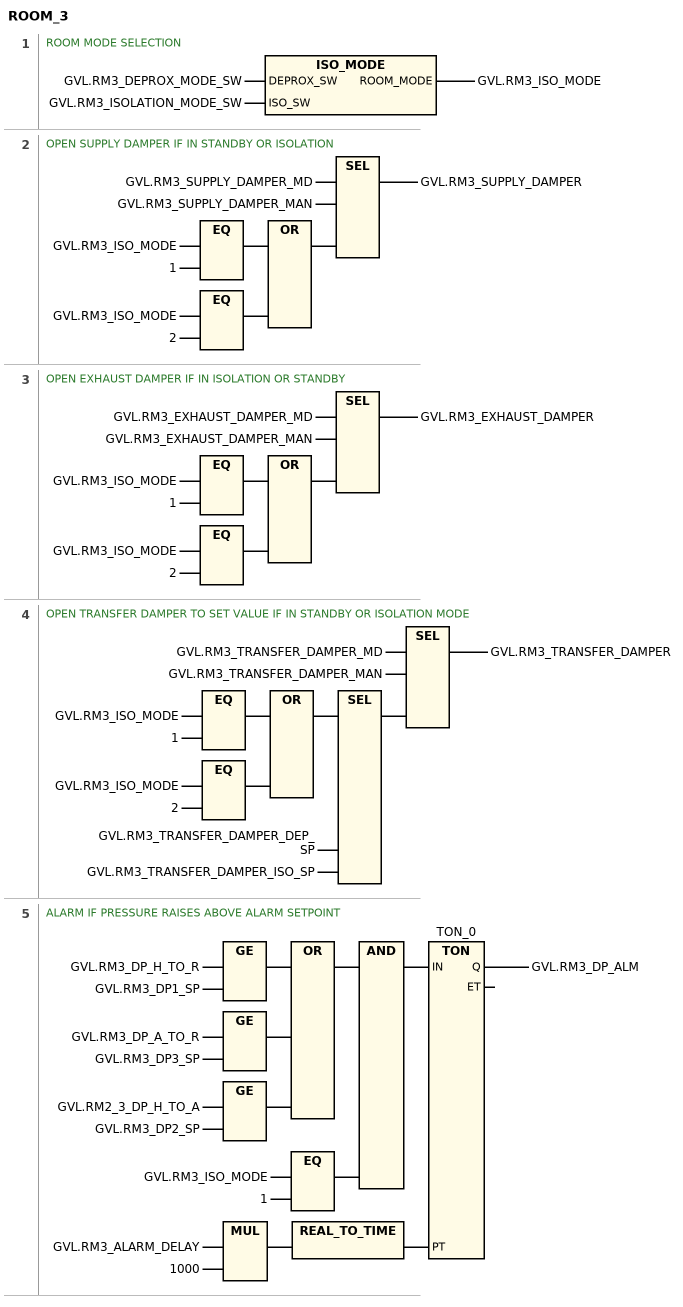
// NETWORK 1
// ROOM MODE SELECTION
ISO_MODE(DEPROX_SW := GVL.RM3_DEPROX_MODE_SW, ISO_SW := GVL.RM3_ISOLATION_MODE_SW);
GVL.RM3_ISO_MODE := ISO_MODE.ROOM_MODE;

// NETWORK 2
// OPEN SUPPLY DAMPER IF IN STANDBY OR ISOLATION
GVL.RM3_SUPPLY_DAMPER := SEL(GVL.RM3_SUPPLY_DAMPER_MD, GVL.RM3_SUPPLY_DAMPER_MAN, GVL.RM3_ISO_MODE = 1 OR GVL.RM3_ISO_MODE = 2);

// NETWORK 3
// OPEN EXHAUST DAMPER IF IN ISOLATION OR STANDBY
GVL.RM3_EXHAUST_DAMPER := SEL(GVL.RM3_EXHAUST_DAMPER_MD, GVL.RM3_EXHAUST_DAMPER_MAN, GVL.RM3_ISO_MODE = 1 OR GVL.RM3_ISO_MODE = 2);

// NETWORK 4
// OPEN TRANSFER DAMPER TO SET VALUE IF IN STANDBY OR ISOLATION MODE
GVL.RM3_TRANSFER_DAMPER := SEL(GVL.RM3_TRANSFER_DAMPER_MD, GVL.RM3_TRANSFER_DAMPER_MAN, SEL(GVL.RM3_ISO_MODE = 1 OR GVL.RM3_ISO_MODE = 2, GVL.RM3_TRANSFER_DAMPER_DEP_SP, GVL.RM3_TRANSFER_DAMPER_ISO_SP));

// NETWORK 5
// ALARM IF PRESSURE RAISES ABOVE ALARM SETPOINT
TON_0(IN := (GVL.RM3_DP_H_TO_R >= GVL.RM3_DP1_SP OR GVL.RM3_DP_A_TO_R >= GVL.RM3_DP3_SP OR GVL.RM2_3_DP_H_TO_A >= GVL.RM3_DP2_SP) AND GVL.RM3_ISO_MODE = 1, PT := REAL_TO_TIME(GVL.RM3_ALARM_DELAY * 1000)); // TON
GVL.RM3_DP_ALM := TON_0.Q;

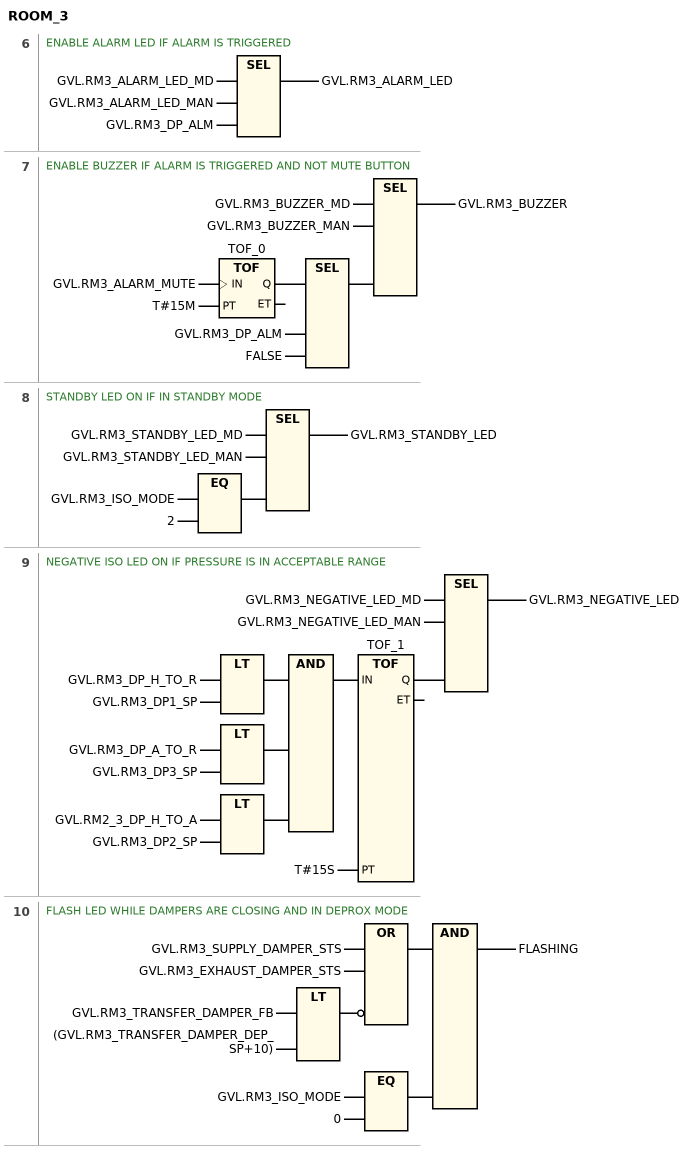
// NETWORK 6
// ENABLE ALARM LED IF ALARM IS TRIGGERED
GVL.RM3_ALARM_LED := SEL(GVL.RM3_ALARM_LED_MD, GVL.RM3_ALARM_LED_MAN, GVL.RM3_DP_ALM);

// NETWORK 7
// ENABLE BUZZER IF ALARM IS TRIGGERED AND NOT MUTE BUTTON
_rt1(CLK := GVL.RM3_ALARM_MUTE);
TOF_0(IN := _rt1.Q, PT := T#15M); // TOF
GVL.RM3_BUZZER := SEL(GVL.RM3_BUZZER_MD, GVL.RM3_BUZZER_MAN, SEL(TOF_0.Q, GVL.RM3_DP_ALM, FALSE));

// NETWORK 8
// STANDBY LED ON IF IN STANDBY MODE
GVL.RM3_STANDBY_LED := SEL(GVL.RM3_STANDBY_LED_MD, GVL.RM3_STANDBY_LED_MAN, GVL.RM3_ISO_MODE = 2);

// NETWORK 9
// NEGATIVE ISO LED ON IF PRESSURE IS IN ACCEPTABLE RANGE
TOF_1(IN := GVL.RM3_DP_H_TO_R < GVL.RM3_DP1_SP AND GVL.RM3_DP_A_TO_R < GVL.RM3_DP3_SP AND GVL.RM2_3_DP_H_TO_A < GVL.RM3_DP2_SP, PT := T#15S); // TOF
GVL.RM3_NEGATIVE_LED := SEL(GVL.RM3_NEGATIVE_LED_MD, GVL.RM3_NEGATIVE_LED_MAN, TOF_1.Q);

// NETWORK 10
// FLASH LED WHILE DAMPERS ARE CLOSING AND IN DEPROX MODE
FLASHING := (GVL.RM3_SUPPLY_DAMPER_STS OR GVL.RM3_EXHAUST_DAMPER_STS OR NOT (GVL.RM3_TRANSFER_DAMPER_FB < ((GVL.RM3_TRANSFER_DAMPER_DEP_SP+10)))) AND GVL.RM3_ISO_MODE = 0;

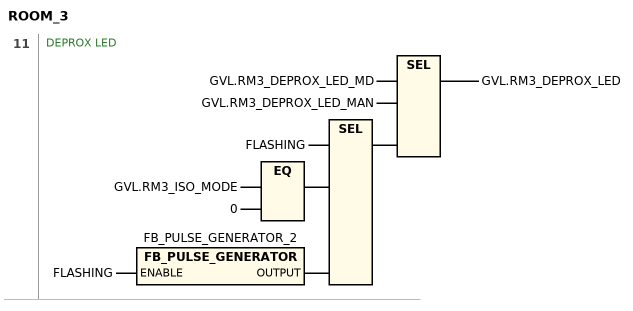
// NETWORK 11
// DEPROX LED
FB_PULSE_GENERATOR_2(ENABLE := FLASHING); // FB_PULSE_GENERATOR
GVL.RM3_DEPROX_LED := SEL(GVL.RM3_DEPROX_LED_MD, GVL.RM3_DEPROX_LED_MAN, SEL(FLASHING, GVL.RM3_ISO_MODE = 0, FB_PULSE_GENERATOR_2.OUTPUT));

END_PROGRAM

// DCCM_PCL_2/Application/ROOM_4
PROGRAM ROOM_4
VAR
	TON_0: TON;
	TOF_0: TOF;
	TOF_1: TOF;
	FLASHING: BOOL;
	FB_PULSE_GENERATOR_1: FB_PULSE_GENERATOR;
END_VAR
VAR // added by the converter: edge detectors and wires of the graphical bodies
    _rt1 : R_TRIG;
END_VAR

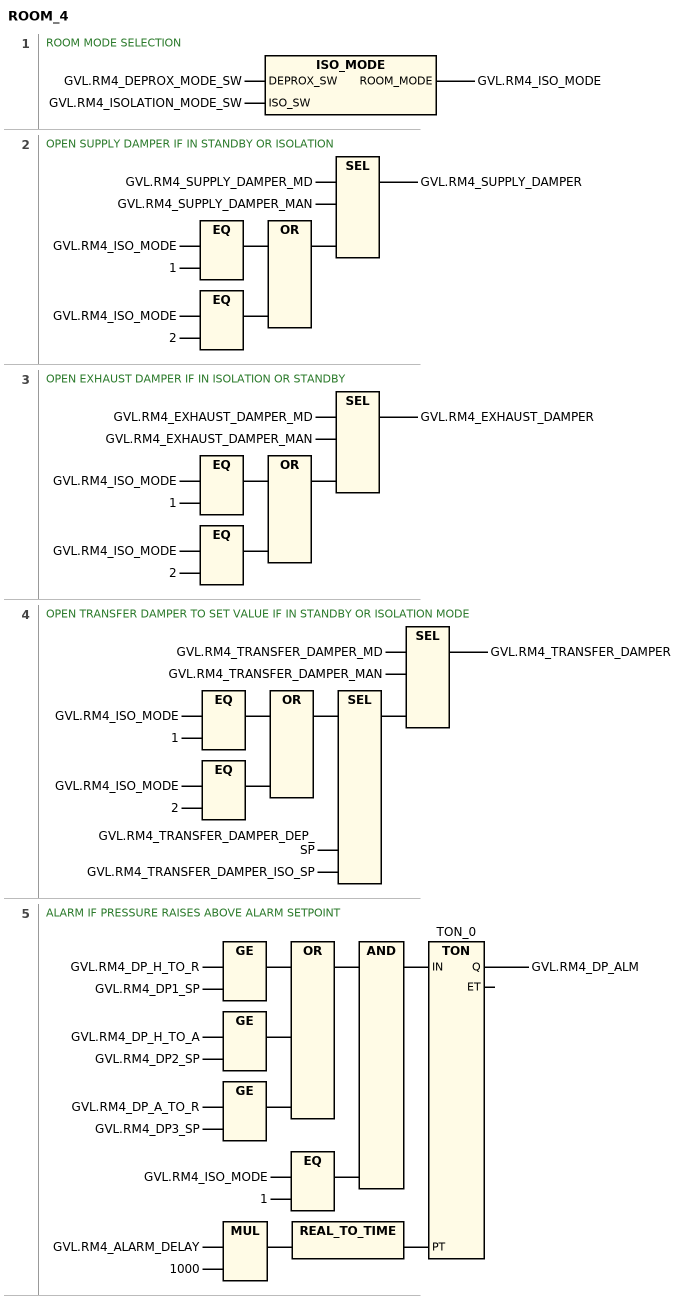
// NETWORK 1
// ROOM MODE SELECTION
ISO_MODE(DEPROX_SW := GVL.RM4_DEPROX_MODE_SW, ISO_SW := GVL.RM4_ISOLATION_MODE_SW);
GVL.RM4_ISO_MODE := ISO_MODE.ROOM_MODE;

// NETWORK 2
// OPEN SUPPLY DAMPER IF IN STANDBY OR ISOLATION
GVL.RM4_SUPPLY_DAMPER := SEL(GVL.RM4_SUPPLY_DAMPER_MD, GVL.RM4_SUPPLY_DAMPER_MAN, GVL.RM4_ISO_MODE = 1 OR GVL.RM4_ISO_MODE = 2);

// NETWORK 3
// OPEN EXHAUST DAMPER IF IN ISOLATION OR STANDBY
GVL.RM4_EXHAUST_DAMPER := SEL(GVL.RM4_EXHAUST_DAMPER_MD, GVL.RM4_EXHAUST_DAMPER_MAN, GVL.RM4_ISO_MODE = 1 OR GVL.RM4_ISO_MODE = 2);

// NETWORK 4
// OPEN TRANSFER DAMPER TO SET VALUE IF IN STANDBY OR ISOLATION MODE
GVL.RM4_TRANSFER_DAMPER := SEL(GVL.RM4_TRANSFER_DAMPER_MD, GVL.RM4_TRANSFER_DAMPER_MAN, SEL(GVL.RM4_ISO_MODE = 1 OR GVL.RM4_ISO_MODE = 2, GVL.RM4_TRANSFER_DAMPER_DEP_SP, GVL.RM4_TRANSFER_DAMPER_ISO_SP));

// NETWORK 5
// ALARM IF PRESSURE RAISES ABOVE ALARM SETPOINT
TON_0(IN := (GVL.RM4_DP_H_TO_R >= GVL.RM4_DP1_SP OR GVL.RM4_DP_H_TO_A >= GVL.RM4_DP2_SP OR GVL.RM4_DP_A_TO_R >= GVL.RM4_DP3_SP) AND GVL.RM4_ISO_MODE = 1, PT := REAL_TO_TIME(GVL.RM4_ALARM_DELAY * 1000)); // TON
GVL.RM4_DP_ALM := TON_0.Q;

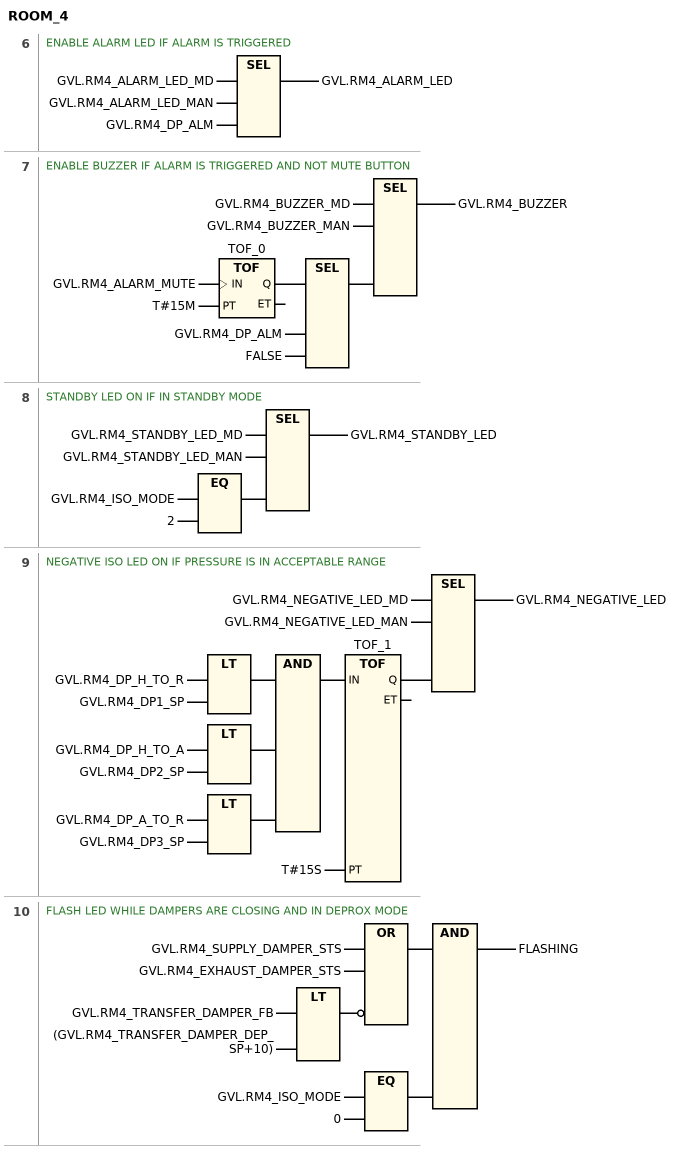
// NETWORK 6
// ENABLE ALARM LED IF ALARM IS TRIGGERED
GVL.RM4_ALARM_LED := SEL(GVL.RM4_ALARM_LED_MD, GVL.RM4_ALARM_LED_MAN, GVL.RM4_DP_ALM);

// NETWORK 7
// ENABLE BUZZER IF ALARM IS TRIGGERED AND NOT MUTE BUTTON
_rt1(CLK := GVL.RM4_ALARM_MUTE);
TOF_0(IN := _rt1.Q, PT := T#15M); // TOF
GVL.RM4_BUZZER := SEL(GVL.RM4_BUZZER_MD, GVL.RM4_BUZZER_MAN, SEL(TOF_0.Q, GVL.RM4_DP_ALM, FALSE));

// NETWORK 8
// STANDBY LED ON IF IN STANDBY MODE
GVL.RM4_STANDBY_LED := SEL(GVL.RM4_STANDBY_LED_MD, GVL.RM4_STANDBY_LED_MAN, GVL.RM4_ISO_MODE = 2);

// NETWORK 9
// NEGATIVE ISO LED ON IF PRESSURE IS IN ACCEPTABLE RANGE
TOF_1(IN := GVL.RM4_DP_H_TO_R < GVL.RM4_DP1_SP AND GVL.RM4_DP_H_TO_A < GVL.RM4_DP2_SP AND GVL.RM4_DP_A_TO_R < GVL.RM4_DP3_SP, PT := T#15S); // TOF
GVL.RM4_NEGATIVE_LED := SEL(GVL.RM4_NEGATIVE_LED_MD, GVL.RM4_NEGATIVE_LED_MAN, TOF_1.Q);

// NETWORK 10
// FLASH LED WHILE DAMPERS ARE CLOSING AND IN DEPROX MODE
FLASHING := (GVL.RM4_SUPPLY_DAMPER_STS OR GVL.RM4_EXHAUST_DAMPER_STS OR NOT (GVL.RM4_TRANSFER_DAMPER_FB < ((GVL.RM4_TRANSFER_DAMPER_DEP_SP+10)))) AND GVL.RM4_ISO_MODE = 0;

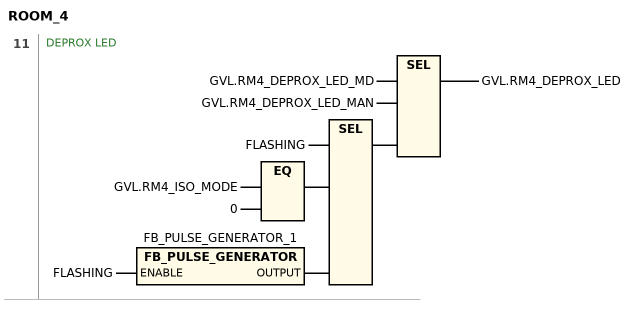
// NETWORK 11
// DEPROX LED
FB_PULSE_GENERATOR_1(ENABLE := FLASHING); // FB_PULSE_GENERATOR
GVL.RM4_DEPROX_LED := SEL(GVL.RM4_DEPROX_LED_MD, GVL.RM4_DEPROX_LED_MAN, SEL(FLASHING, GVL.RM4_ISO_MODE = 0, FB_PULSE_GENERATOR_1.OUTPUT));

END_PROGRAM

// DCCM_PCL_2/Application/OUTPUT_MAPPING
PROGRAM OUTPUT_MAPPING
VAR
		voltage_converter: FB_0_10V_TO_2_10V_OUTPUT;
END_VAR

//MAPPING MEMORY WORDS TO HARDWARE OUTPUTS

//qRM1_TRANSFER_DAMPER := TO_INT(GVL.RM1_TRANSFER_DAMPER) * 100;								//MODULE 1 TM3AQ4 OUTPUT 0
//qRM2_TRANSFER_DAMPER := TO_INT(GVL.RM2_TRANSFER_DAMPER) * 100;								//MODULE 1 TM3AQ4 OUTPUT 1
//qRM3_TRANSFER_DAMPER := TO_INT(GVL.RM3_TRANSFER_DAMPER) * 100;								//MODULE 1 TM3AQ4 OUTPUT 2
//qRM4_TRANSFER_DAMPER := TO_INT(GVL.RM4_TRANSFER_DAMPER) * 100;								//MODULE 1 TM3AQ4 OUTPUT 3

voltage_converter(IN_PRCT := GVL.RM1_TRANSFER_DAMPER);
qRM1_TRANSFER_DAMPER := TO_INT((120-voltage_converter.OUT_PRCT)*100); //AI0  0v=open 10v=close

voltage_converter(IN_PRCT := GVL.RM2_TRANSFER_DAMPER);
qRM2_TRANSFER_DAMPER := TO_INT((120-voltage_converter.OUT_PRCT)*100); //AI0  0v=open 10v=close

voltage_converter(IN_PRCT := GVL.RM3_TRANSFER_DAMPER);
qRM3_TRANSFER_DAMPER := TO_INT((120-voltage_converter.OUT_PRCT)*100); //AI0  0v=open 10v=close

voltage_converter(IN_PRCT := GVL.RM4_TRANSFER_DAMPER);
qRM4_TRANSFER_DAMPER := TO_INT((120-voltage_converter.OUT_PRCT)*100); //AI0  0v=open 10v=close

qRM1_SUPPLY_DAMPER := NOT GVL.RM1_SUPPLY_DAMPER;												//MODULE 5 TM3DM24R OUTPUT 0
qRM2_SUPPLY_DAMPER := NOT GVL.RM2_SUPPLY_DAMPER;												//MODULE 5 TM3DM24R OUTPUT 1
qRM3_SUPPLY_DAMPER := NOT GVL.RM3_SUPPLY_DAMPER;												//MODULE 5 TM3DM24R OUTPUT 2
qRM4_SUPPLY_DAMPER := NOT GVL.RM4_SUPPLY_DAMPER;												//MODULE 5 TM3DM24R OUTPUT 3

qRM1_EXHAUST_DAMPER := NOT GVL.RM1_EXHAUST_DAMPER;												//MODULE 5 TM3DM24R OUTPUT 4
qRM2_EXHAUST_DAMPER := NOT GVL.RM2_EXHAUST_DAMPER;												//MODULE 5 TM3DM24R OUTPUT 5
qRM3_EXHAUST_DAMPER := NOT GVL.RM3_EXHAUST_DAMPER;												//MODULE 5 TM3DM24R OUTPUT 6
qRM4_EXHAUST_DAMPER := NOT GVL.RM4_EXHAUST_DAMPER;												//MODULE 5 TM3DM24R OUTPUT 7

qRM1_NEGATIVE_LED := GVL.RM1_NEGATIVE_LED;													//MODULE 6 TM3DM24R OUTPUT 0
qRM1_DEPROX_LED := GVL.RM1_DEPROX_LED;														//MODULE 6 TM3DM24R OUTPUT 1
qRM1_ALARM_LED := GVL.RM1_ALARM_LED;														//MODULE 6 TM3DM24R OUTPUT 2
qRM1_STANDBY_LED := GVL.RM1_STANDBY_LED;													//MODULE 6 TM3DM24R OUTPUT 3
qRM2_NEGATIVE_LED := GVL.RM2_NEGATIVE_LED;													//MODULE 6 TM3DM24R OUTPUT 4
qRM2_DEPROX_LED := GVL.RM2_DEPROX_LED;														//MODULE 6 TM3DM24R OUTPUT 5
qRM2_ALARM_LED := GVL.RM2_ALARM_LED;														//MODULE 6 TM3DM24R OUTPUT 6
qRM2_STANDBY_LED := GVL.RM2_STANDBY_LED;													//MODULE 6 TM3DM24R OUTPUT 7

qRM3_NEGATIVE_LED := GVL.RM3_NEGATIVE_LED;													//MODULE 7 TM3DQ16R OUTPUT 0
qRM3_DEPROX_LED := GVL.RM3_DEPROX_LED;														//MODULE 7 TM3DQ16R OUTPUT 1
qRM3_ALARM_LED := GVL.RM3_ALARM_LED;														//MODULE 7 TM3DQ16R OUTPUT 2
qRM3_STANDBY_LED := GVL.RM3_STANDBY_LED;													//MODULE 7 TM3DQ16R OUTPUT 3
qRM4_NEGATIVE_LED := GVL.RM4_NEGATIVE_LED;													//MODULE 7 TM3DQ16R OUTPUT 4
qRM4_DEPROX_LED := GVL.RM4_DEPROX_LED;														//MODULE 7 TM3DQ16R OUTPUT 5
qRM4_ALARM_LED := GVL.RM4_ALARM_LED;														//MODULE 7 TM3DQ16R OUTPUT 6
qRM4_STANDBY_LED := GVL.RM4_STANDBY_LED;													//MODULE 7 TM3DQ16R OUTPUT 7
qRM1_BUZZER := GVL.RM1_BUZZER;																//MODULE 7 TM3DQ16R OUTPUT 8
qRM2_BUZZER := GVL.RM2_BUZZER;																//MODULE 7 TM3DQ16R OUTPUT 9
qRM3_BUZZER := GVL.RM3_BUZZER;																//MODULE 7 TM3DQ16R OUTPUT 10
qRM4_BUZZER := GVL.RM4_BUZZER;																//MODULE 7 TM3DQ16R OUTPUT 11

GVL.DEPROX_TOTAL:= 4;//BOOL_TO_REAL(GVL.RM3_DEPROX_MODE_SW)+BOOL_TO_REAL(GVL.RM2_DEPROX_MODE_SW)+BOOL_TO_REAL(GVL.RM1_DEPROX_MODE_SW)+BOOL_TO_REAL(GVL.RM4_DEPROX_MODE_SW);

END_PROGRAM

// DCCM_PCL_2/Application/SR_Main
PROGRAM SR_Main
VAR
END_VAR

// NETWORK 1

END_PROGRAM

// DCCM_PCL_2/Application/FBs/DUTY
FUNCTION_BLOCK DUTY
VAR_INPUT
	DUTY_MAN: BOOL;
	DUTY_MD: BOOL;
	TOGGLE: BOOL;
END_VAR
VAR_OUTPUT
	DUTY: BOOL;
END_VAR

IF (TOGGLE AND DUTY = TRUE AND DUTY_MD = FALSE) THEN
	DUTY := FALSE;
ELSIF (TOGGLE AND DUTY = FALSE AND DUTY_MD = FALSE) THEN
	DUTY := TRUE;
ELSE
	DUTY := DUTY_MAN;
END_IF

END_FUNCTION_BLOCK

// DCCM_PCL_2/Application/FBs/DUTY_CHANGE
FUNCTION_BLOCK DUTY_CHANGE
VAR_INPUT
	INPUT: BOOL;
END_VAR
VAR_OUTPUT
	NEW_DUTY: BOOL;
END_VAR
VAR_INPUT
	CURRENT_DUTY: BOOL;
END_VAR

IF INPUT THEN
	IF CURRENT_DUTY = 1 THEN
		NEW_DUTY := 0;
	ELSIF CURRENT_DUTY = 0 THEN
		NEW_DUTY := 1;
	END_IF
END_IF

END_FUNCTION_BLOCK

// DCCM_PCL_2/Application/FBs/FB_9StatesMonitoring
FUNCTION_BLOCK FB_9StatesMonitoring
VAR
	ENABLE_OFF: BOOL := FALSE;
	ENABLE_ON: BOOL := FALSE;
	STATUS_ON: BOOL := FALSE;
	STATUS_OFF: BOOL := FALSE;
	FIRE_ON: BOOL := FALSE;
	FIRE_OFF: BOOL := FALSE;
	BEEN_RUNNING_OK: BOOL := FALSE;
	NOT_BEEN_RUNNING_OK: BOOL := FALSE;
	ALL_OFF: BOOL := FALSE;
	NOT_ALL_OFF: BOOL := FALSE;
	START_DELAY_ON: BOOL := FALSE;
	START_DELAY_OFF: BOOL := FALSE;
	STOP_DELAY_ON: BOOL := FALSE;
	STOP_DELAY_OFF: BOOL := FALSE;
	ENABLE_TIMER_ON: BOOL := FALSE;
	ENABLE_TIMER_OFF: BOOL := FALSE;
	BEEN_RUNNING_OK_LATCH: RS;
	ALL_OFF_LATCH: RS;
	START_DELAY_TON: TON;
	STOP_DELAY_TON: TON;
	STOPPED: INT;
END_VAR
VAR_INPUT
	ENABLE: BOOL := FALSE;
	STATUS: BOOL := FALSE;
	FIRE: BOOL := FALSE;
END_VAR
VAR_OUTPUT
	STATE: ET_9STATE_MONITORING := 9;
END_VAR

(* 
Version 1.0
Last Updated: 28/01/2020

9 States Monitoring. Value from 0 to 9
	STOPPED := 0,
	RUNNING := 1,
	STARTING := 2,
	STOPPING := 3,
	START_FAIL := 4,
	STOP_FAIL := 5,
	UNEXPECTED_START := 6,
	UNEXPECTED_STOP := 7,
	FIRE_STOP := 8,
	UNKNOWN := 9
*)

ENABLE_OFF := (ENABLE = FALSE);
ENABLE_ON := (ENABLE = TRUE);
STATUS_ON := (STATUS = TRUE);
STATUS_OFF := (STATUS = FALSE);
FIRE_ON := (FIRE = TRUE);
FIRE_OFF := (FIRE = FALSE);

BEEN_RUNNING_OK_LATCH(SET := ENABLE_ON AND STATUS_ON, RESET1 := ENABLE_OFF);
BEEN_RUNNING_OK := BEEN_RUNNING_OK_LATCH.Q1;

ALL_OFF_LATCH(SET := ENABLE_OFF AND STATUS_OFF, RESET1 := ENABLE_ON);
ALL_OFF := ALL_OFF_LATCH.Q1;

START_DELAY_TON(IN := ENABLE_ON, PT := T#30S);
START_DELAY_ON := START_DELAY_TON.Q;

STOP_DELAY_TON(IN := ENABLE_OFF, PT := T#30S);
STOP_DELAY_ON := STOP_DELAY_TON.Q;

ENABLE_TIMER_ON := ((START_DELAY_TON.ET < T#30S AND ENABLE_ON) OR (STOP_DELAY_TON.ET < T#30S AND ENABLE_OFF));

START_DELAY_OFF := NOT START_DELAY_ON;
STOP_DELAY_OFF := NOT STOP_DELAY_ON;
ENABLE_TIMER_OFF := NOT ENABLE_TIMER_ON;
NOT_BEEN_RUNNING_OK := NOT BEEN_RUNNING_OK;
NOT_ALL_OFF := NOT ALL_OFF;

IF (ENABLE_ON AND STATUS_OFF AND FIRE_ON) THEN
	STATE := ET_9STATE_MONITORING.FIRE_STOP;
ELSIF (ENABLE_OFF AND STATUS_ON AND STOP_DELAY_ON AND NOT_BEEN_RUNNING_OK AND NOT_ALL_OFF) THEN
	STATE := ET_9STATE_MONITORING.STOP_FAIL;
ELSIF (ENABLE_ON AND STATUS_OFF AND START_DELAY_ON AND NOT_BEEN_RUNNING_OK AND NOT_ALL_OFF) THEN
	STATE := ET_9STATE_MONITORING.START_FAIL;
ELSIF (ENABLE_OFF AND STATUS_ON AND ENABLE_TIMER_OFF AND STOP_DELAY_ON AND ENABLE_TIMER_OFF AND ALL_OFF) THEN
	STATE := ET_9STATE_MONITORING.UNEXPECTED_START;
ELSIF (ENABLE_ON AND STATUS_OFF AND START_DELAY_ON AND FIRE_OFF AND ENABLE_TIMER_OFF AND BEEN_RUNNING_OK AND NOT_ALL_OFF) THEN
	STATE := ET_9STATE_MONITORING.UNEXPECTED_STOP;
ELSIF (ENABLE_OFF AND STATUS_ON AND ENABLE_TIMER_ON AND STOP_DELAY_OFF AND FIRE_OFF) THEN
	STATE := ET_9STATE_MONITORING.STOPPING;
ELSIF (ENABLE_ON AND STATUS_ON) THEN
	STATE := ET_9STATE_MONITORING.RUNNING;
ELSIF (ENABLE_ON AND STATUS_OFF AND ENABLE_TIMER_ON AND START_DELAY_OFF AND FIRE_OFF) THEN
	STATE := ET_9STATE_MONITORING.STARTING;
ELSIF (ENABLE_OFF AND STATUS_OFF) THEN
	STATE := ET_9STATE_MONITORING.STOPPED;
ELSE
	STATE := ET_9STATE_MONITORING.UNKNOWN;
END_IF;

END_FUNCTION_BLOCK

// DCCM_PCL_2/Application/FBs/FB_DUTY_DUTY_STANDBY_PUMP_SPD
FUNCTION_BLOCK FB_DUTY_DUTY_STANDBY_PUMP_SPD
VAR_INPUT
	SPD_DEM: REAL;
	P1_FLT: BOOL;
	P2_FLT: BOOL;
	P3_FLT: BOOL;
	DUTY: INT;
END_VAR
VAR_OUTPUT
	PUMP1_SPD: REAL;
	PUMP2_SPD: REAL;
	PUMP3_SPD: REAL;
END_VAR

IF (P1_FLT = TRUE AND P2_FLT = TRUE AND P3_FLT = TRUE) THEN				// IF ALL PUMPS IN FAULT, REDUCE SPEED TO 0 FOR ALL PUMPS
	PUMP1_SPD := 0;
	PUMP2_SPD := 0;
	PUMP3_SPD := 0;
ELSIF (DUTY = 0 AND P1_FLT = FALSE AND P2_FLT = FALSE) THEN				//IF PUMP 1 DUTY
	PUMP1_SPD := LIMIT(0, SPD_DEM, 100);
	PUMP2_SPD := LIMIT(0, SPD_DEM - 100, 100);
	PUMP3_SPD := 0;
ELSIF (DUTY = 1 AND P2_FLT = FALSE AND P3_FLT = FALSE)THEN				//IF PUMP 2 DUTY
	PUMP2_SPD := LIMIT(0, SPD_DEM, 100);
	PUMP3_SPD := LIMIT(0, SPD_DEM - 100, 100);
	PUMP1_SPD := 0;
ELSIF(DUTY = 2 AND P3_FLT = FALSE AND P1_FLT = FALSE) THEN				//IF PUMP 3 DUTY
	PUMP3_SPD := LIMIT(0, SPD_DEM, 100);
	PUMP1_SPD := LIMIT(0, SPD_DEM - 100, 100);
	PUMP2_SPD := 0;	
ELSIF (DUTY = 0 AND P1_FLT = TRUE AND P2_FLT = FALSE) THEN				//IF PUMP 1 DUTY AND PUMP 1 IS IN FAULT
	PUMP3_SPD := LIMIT(0, SPD_DEM, 100);
	PUMP2_SPD := LIMIT(0, SPD_DEM - 100, 100);
	PUMP1_SPD := 0;
ELSIF (DUTY = 0 AND P1_FLT = FALSE AND P2_FLT = TRUE) THEN				// IF PUMP 1 DUTY AND PUMP 2 IS IN FAULT
	PUMP1_SPD := LIMIT(0, SPD_DEM, 100);
	PUMP3_SPD := LIMIT(0, SPD_DEM - 100, 100);
	PUMP2_SPD := 0;
ELSIF (DUTY = 0 AND P1_FLT = TRUE AND P2_FLT = TRUE) THEN				//IF PUMP 1 DUTY AND PUMP 1 & 2 ARE IN FAULT
	PUMP3_SPD := LIMIT(0, SPD_DEM, 100);
	PUMP1_SPD := 0;
	PUMP2_SPD := 0;
ELSIF (DUTY = 1 AND P2_FLT = TRUE AND P3_FLT = FALSE) THEN				//IF PUMP 2 DUTY AND PUMP 2 IS IN FAULT
	PUMP1_SPD := LIMIT(0, SPD_DEM, 100);
	PUMP3_SPD := LIMIT(0, SPD_DEM - 100, 100);
	PUMP2_SPD := 0;
ELSIF (DUTY = 1 AND P2_FLT = FALSE AND P3_FLT := TRUE) THEN				//IF PUMP 2 DUTY AND PUMP 3 IS IN FAULT
	PUMP2_SPD := LIMIT(0, SPD_DEM, 100);
	PUMP1_SPD := LIMIT(0, SPD_DEM - 100, 100);
	PUMP3_SPD := 0;
ELSIF (DUTY = 1 AND P2_FLT = TRUE AND P3_FLT := TRUE) THEN				//IF PUMP 2 DUTY AND PUMP 2 & 3 ARE IN FAULT
	PUMP1_SPD := LIMIT(0, SPD_DEM, 100);
	PUMP2_SPD := 0;
	PUMP3_SPD := 0;
ELSIF (DUTY = 2 AND P3_FLT = TRUE AND P1_FLT = FALSE) THEN				//IF PUMP 3 DUTY AND PUMP 3 IS IN FAULT 
	PUMP2_SPD := LIMIT(0, SPD_DEM, 100);
	PUMP1_SPD := LIMIT(0, SPD_DEM - 100, 100);
	PUMP3_SPD := 0;
ELSIF (DUTY = 2 AND P3_FLT = FALSE AND P1_FLT = TRUE) THEN				//IF PUMP 3 DUTY AND PUMP 1 IS IN FAULT
	PUMP3_SPD := LIMIT(0, SPD_DEM, 100);
	PUMP2_SPD := LIMIT(0, SPD_DEM - 100, 100);
	PUMP1_SPD := 0;
ELSIF (DUTY = 2 AND P3_FLT = TRUE AND P1_FLT = TRUE) THEN				//IF PUMP 3 DUTY AND PUMP 3 & 1 ARE IN FAULT
	PUMP2_SPD := LIMIT(0, SPD_DEM, 100);
	PUMP3_SPD := 0;
	PUMP1_SPD := 0;
END_IF

END_FUNCTION_BLOCK

// DCCM_PCL_2/Application/FBs/FB_FLOATING_VALVE
FUNCTION_BLOCK FB_FLOATING_VALVE
VAR_INPUT
	VALVE_OUTPUT: REAL;
	VALVE_TIME: TIME;
END_VAR
VAR_OUTPUT
	VALVE_OPEN: BOOL;
	VALVE_CLOSE: BOOL;
END_VAR
VAR
	CURRENT_POS: REAL;
	MOVE_TIME: TIME;
	MOVE_POS: REAL;
	RS_0: RS;
	TON1: TON;
	OPEN_STOP: BOOL;
	TON2: TON;
	CLOSE_STOP: BOOL;
	RS_1: RS;
END_VAR

IF (VALVE_OUTPUT > CURRENT_POS) THEN
	MOVE_POS := VALVE_OUTPUT - CURRENT_POS;
 	MOVE_TIME := TO_TIME(TO_REAL(VALVE_TIME) * (MOVE_POS / 100)); 
	VALVE_OPEN := TRUE;
	TON1(IN := VALVE_OPEN, PT := MOVE_TIME);
	OPEN_STOP := TON1.Q;
	//RS_0(SET := VALVE_OPEN, RESET1 := OPEN_STOP);
	IF (OPEN_STOP = TRUE) THEN
		VALVE_OPEN := FALSE;
		CURRENT_POS := VALVE_OUTPUT;
	END_IF  
ELSIF (VALVE_OUTPUT < CURRENT_POS) THEN
	MOVE_POS := CURRENT_POS - VALVE_OUTPUT;
	MOVE_TIME := TO_TIME(TO_REAL(VALVE_TIME) * (MOVE_POS / 100));
	VALVE_CLOSE := TRUE;
	TON2(IN := VALVE_CLOSE, PT := MOVE_TIME);
	CLOSE_STOP := TON2.Q;
	//RS_1(SET := VALVE_OPEN, RESET1 := CLOSE_STOP);
	IF (CLOSE_STOP = TRUE) THEN
		VALVE_CLOSE := FALSE;
		CURRENT_POS := VALVE_OUTPUT;
	END_IF
ELSE
	VALVE_OPEN := FALSE;
	VALVE_CLOSE := FALSE;
END_IF

END_FUNCTION_BLOCK

// DCCM_PCL_2/Application/FBs/FB_HEATING_OR_COOLING
FUNCTION_BLOCK FB_HEATING_OR_COOLING
VAR_INPUT
	SAT: REAL;
	SATSP: REAL;
	DB: REAL;
END_VAR
VAR_OUTPUT
	ENABLE_HEATING: BOOL;
	ENABLE_COOLING: BOOL;
END_VAR
VAR_INPUT
	RUN: BOOL;
	HV: REAL;
	CV: REAL;
END_VAR

IF (SAT >= (SATSP + DB) AND RUN AND HV = 0) THEN
	ENABLE_COOLING := TRUE AND ENABLE_HEATING := FALSE;
ELSIF (SAT <= (SATSP - DB) AND RUN AND CV = 0) THEN
	ENABLE_COOLING := FALSE AND ENABLE_HEATING := TRUE;
ELSE
	ENABLE_COOLING := FALSE AND ENABLE_HEATING := FALSE;	
END_IF

END_FUNCTION_BLOCK

// DCCM_PCL_2/Application/FBs/FB_OMODE
FUNCTION_BLOCK FB_OMODE
VAR_INPUT
	ENABLE_BY_TP: BOOL;
	ENABLE_BY_PIR: BOOL;
	ENABLE_BY_AHRS: BOOL;
	MODE: BOOL;
	OMODE_MANUAL: ET_OMODE;
	TPTYPE: BOOL;
END_VAR
VAR_OUTPUT
	OMODE: ET_OMODE;
END_VAR




IF (MODE) THEN
	IF (ENABLE_BY_TP) THEN				//AUTO MODE
		OMODE := ET_OMODE.SCH;
	ELSIF (ENABLE_BY_AHRS) THEN
		OMODE := ET_OMODE.AHRS;
	ELSIF (ENABLE_BY_PIR) THEN
		OMODE := ET_OMODE.MOTDETECT;
	ELSIF (TPTYPE) THEN
		OMODE := ET_OMODE.UNOCC;
	ELSE
		OMODE := ET_OMODE.SETBACK;
	END_IF
ELSE
	OMODE := OMODE_MANUAL;				//MANUAL MODE
END_IF

END_FUNCTION_BLOCK

// DCCM_PCL_2/Application/FBs/FB_PMODE
FUNCTION_BLOCK FB_PMODE
VAR_INPUT
	OMODE: ET_OMODE;
	IS_NOT_SMOKE: BOOL := TRUE;
	FIRE: BOOL;
	PCMS_SIGNAL: INT;
	PCMS_PRIMARY: INT;
	PCMS_MODE: BOOL := TRUE;
	IS_DAMPER_LOCK: BOOL;
	IS_DAMPER_RESET: BOOL;
	IS_PURGE_RUN: BOOL;
	IS_DAMPER_STARTED: BOOL;
	PMODE_MODE: BOOL := TRUE;
	PMODE_MANUAL: ET_PMODE;
END_VAR
VAR_OUTPUT
	AHU_ENABLE: BOOL;
	PMODE: ET_PMODE;
END_VAR

(*  
	Version 1.0
	Last modified: 15/8/2022
	Operating theater mode
	PLEASE USE  FOR OPERATING THEATER ONLY
	IT DOES NOT IMPLEMENT UNOCC, OP_START MODE
	
	OFF_NORMAL := 0,
	OFF_PCMS := 1,
	OFF_FIRE := 2,
	OFF_DMPRLCK := 3,
	OFF_RESET := 4,
	STARTUP := 5,
	RUN_PUR := 6,
	RUN_NORMAL := 7
*)


IF (PMODE_MODE) THEN
	IF (FIRE) THEN
		PMODE := ET_PMODE.OFF_Fire;
	ELSIF (IS_DAMPER_LOCK) THEN
		PMODE := ET_PMODE.OFF_DMPRLOCK;
	ELSIF ((ABS(PCMS_SIGNAL) >= ABS(PCMS_PRIMARY)) AND PCMS_MODE) THEN
		PMODE := ET_PMODE.OFF_PCMS;
	ELSIF (IS_DAMPER_RESET) THEN
		PMODE := ET_PMODE.OFF_RESET;
	ELSIF (IS_PURGE_RUN) THEN
		PMODE := ET_PMODE.Purge;
	ELSIF (IS_DAMPER_STARTED) THEN
		PMODE := ET_PMODE.RUN_NORMAL;
	END_IF
ELSE
	PMODE := PMODE_MANUAL;
END_IF;

AHU_ENABLE := (PMODE = ET_PMODE.Startup OR PMODE = ET_PMODE.Purge OR PMODE = ET_PMODE.RUN_NORMAL) AND IS_NOT_SMOKE = FALSE AND OMODE <> ET_OMODE.UNOCC;

END_FUNCTION_BLOCK

// DCCM_PCL_2/Application/FBs/FB_SETPOINT_MODE
FUNCTION_BLOCK FB_SETPOINT_MODE
VAR_INPUT
	OMODE: ET_OMODE;
	PMODE: ET_PMODE;
	DAY_SP: REAL;
	SETBACK_SP: REAL;
	PURGE_SP: REAL;
END_VAR
VAR_OUTPUT
	RESULT: REAL;
END_VAR

(*
//calculate set point based on plant mode and occupancy mode
	/*
	//occupancy mode
	UNOCC := 0,
	OP_START := 1,
	SCH := 2,
	AHRS := 3,
	MOT_DETECT := 4,
	REVERSE1 := 5,
	REVERSE2 := 6,
	SETBACK := 7,
	
	//plant mode
	OFF_NORMAL := 0,
	OFF_PCMS := 1,
	OFF_FIRE := 2,
	OFF_DMPRLCK := 3,
	OFF_DMPRRESET := 4,
	STARTUP := 5,
	RUN_PUR := 6,
	RUN_NORMAL := 7
	*/
*)

IF (PMODE = ET_PMODE.Purge) THEN
	RESULT := PURGE_SP;
ELSIF ((PMODE = ET_PMODE.RUN_NORMAL) OR (PMODE = ET_PMODE.Startup)) THEN
	IF (OMODE = ET_OMODE.SETBACK) THEN
		RESULT := SETBACK_SP;
	ELSIF(OMODE = ET_OMODE.UNOCC) THEN
		RESULT := 0.0;
	ELSE
		RESULT := DAY_SP;
	END_IF
ELSE
	RESULT := DAY_SP;
END_IF

END_FUNCTION_BLOCK

// DCCM_PCL_2/Application/Library/FB_SETPOINT_RAMPING
FUNCTION_BLOCK FB_SETPOINT_RAMPING
VAR_INPUT
	INPUT: REAL;
	RAMPING_DOWN_TIME_SP: REAL := 10;
	RAMPING_UP_TIME_SP: REAL := 10;
END_VAR
VAR_OUTPUT
	OUTPUT: REAL := 0;
END_VAR
VAR
	TIMER: TON;
	INCREMENT: REAL;
	INPUT_MEMORY: REAL;
END_VAR

(* Set point Ramping up and down *)
IF (OUTPUT = 0) THEN
	OUTPUT := INPUT;
END_IF;

//find the incerement value
IF(INPUT <> INPUT_MEMORY) THEN 
	INPUT_MEMORY := INPUT;	
	IF (INPUT_MEMORY > OUTPUT) THEN
		INCREMENT := (INPUT_MEMORY - OUTPUT)/RAMPING_UP_TIME_SP;
	ELSIF (INPUT_MEMORY < OUTPUT) THEN
		INCREMENT := (INPUT_MEMORY - OUTPUT)/RAMPING_DOWN_TIME_SP;
	ELSE
		INCREMENT := 0;
	END_IF;
END_IF;


IF(INCREMENT <> 0) THEN
	TIMER(IN := NOT TIMER.Q, PT := T#1S);

	IF (TIMER.Q) THEN
		OUTPUT := OUTPUT + INCREMENT;
	END_IF;
	
	IF(OUTPUT > INPUT_MEMORY) AND (INCREMENT > 0) THEN
		//make sure that the output is not over than ouput
		INCREMENT := 0;
		OUTPUT := INPUT_MEMORY;
	ELSIF (OUTPUT < INPUT_MEMORY) AND (INCREMENT < 0) THEN
		//make sure that the output is not less than input
		INCREMENT := 0;
		OUTPUT := INPUT_MEMORY;
	END_IF;
END_IF;

END_FUNCTION_BLOCK

// DCCM_PCL_2/Application/FBs/FB_WATCHDOG
FUNCTION_BLOCK FB_WATCHDOG
VAR_OUTPUT
	LAST_VALUE: INT;
END_VAR
VAR_INPUT
	VALUE: INT;
END_VAR
VAR_OUTPUT
	TIMEOUT: BOOL;
END_VAR
VAR
	START_DELAY_TON: TON;
END_VAR

START_DELAY_TON(IN := (LAST_VALUE = VALUE), PT := T#120S);
TIMEOUT := START_DELAY_TON.Q;

LAST_VALUE := VALUE;

END_FUNCTION_BLOCK

// DCCM_PCL_2/Application/FBs/LINEAR
FUNCTION_BLOCK LINEAR
VAR_INPUT
	INPUT: REAL;
	X1: REAL;
	Y1: REAL;
	X2: REAL;
	Y2: REAL;
END_VAR
VAR
	M: REAL;
END_VAR
VAR_OUTPUT
	OUTPUT: REAL;
END_VAR

// Y1-Y2 = M(X1-X2)
//M = (Y2-Y1)/(X2-X1)

M := (Y2 - Y1) / (X2 - X1);
OUTPUT := (M * (INPUT - X1)) + Y1;

END_FUNCTION_BLOCK

// DCCM_PCL_2/Application/FBs/SATSP_CALC
FUNCTION_BLOCK SATSP_CALC
VAR_INPUT
	SATSP_MID: REAL;
	SATSP_MIN: REAL;
	SATSP_MAX: REAL;
	TL: REAL;
END_VAR
VAR_OUTPUT
	SATSP: REAL;
END_VAR
VAR
	M: REAL;
END_VAR

IF TL > 0 THEN
	M := (SATSP_MID - SATSP_MIN) / 100.0;
	SATSP := (M * (TL)) + SATSP_MIN;
ELSIF TL < 0 THEN
	M := (SATSP_MAX - SATSP_MID) / 100.0;
	SATSP := (M * ABS(TL)) + SATSP_MID;
ELSE
	SATSP := SATSP_MID;
END_IF;

END_FUNCTION_BLOCK

// DCCM_PCL_2/Application/FBs/SB_HEATING_COOLING
FUNCTION_BLOCK SB_HEATING_COOLING
VAR_INPUT
	ENABLE_COOLING: BOOL;
	ENABLE_HEATING: BOOL;
	SATSP: REAL;
	COOLING_SP: REAL;
	HEATING_SP: REAL;
END_VAR
VAR_OUTPUT
	OUT: REAL;
END_VAR
VAR_INPUT
	OMODE: ET_OMODE;
END_VAR

IF (ENABLE_COOLING AND OMODE = ET_OMODE.SETBACK) THEN
	OUT := COOLING_SP;
ELSIF (ENABLE_HEATING AND OMODE = ET_OMODE.SETBACK) THEN
	OUT := HEATING_SP;
ELSE
	OUT := SATSP;
END_IF

END_FUNCTION_BLOCK

// DCCM_PCL_2/Application/FBs/TERMINAL_LOAD
FUNCTION_BLOCK TERMINAL_LOAD
VAR_INPUT
	RMT: REAL;
	RMTSP: REAL;
END_VAR
VAR_OUTPUT
	TL: REAL;
END_VAR
VAR_INPUT
	COOL_TL: REAL;
	HEAT_TL: REAL;
END_VAR

IF (RMTSP > RMT) THEN
	TL := (-1.0 * HEAT_TL);
ELSE
	TL := COOL_TL;	
END_IF;

END_FUNCTION_BLOCK

// DCCM_PCL_2/Application/SendDeprox
PROGRAM SendDeprox
VAR
	My_Read_Var: READ_VAR;
	SEND_Buffer: ARRAY[0..3] OF INT;
	My_Addr_Table: ADDRESS;
	My_Addm: ADDM;
	My_Blink: BLINK;
	My_FLOAT: INT;
	lastValue: INT;
	watchdog: FB_PCMS_WATCHDOG;
	MY_WRITE_VAR: WRITE_VAR;
END_VAR

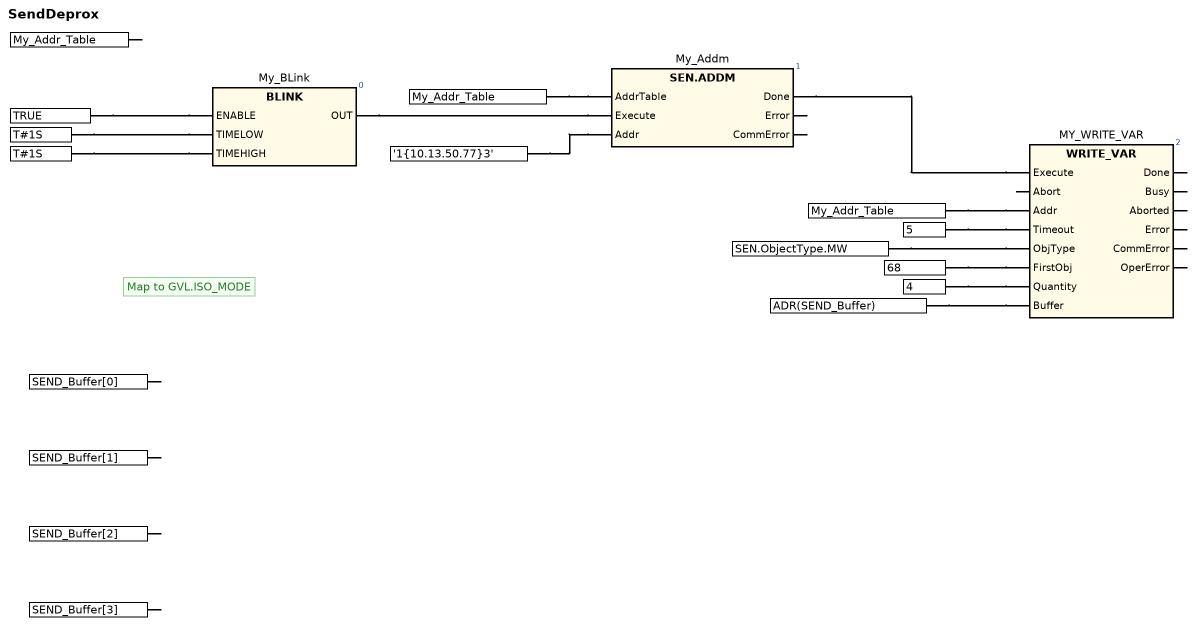
// Map to GVL.ISO_MODE
My_BLink(ENABLE := TRUE, TIMELOW := T#1S, TIMEHIGH := T#1S); // BLINK
My_Addm(AddrTable := My_Addr_Table, Execute := My_BLink.OUT, Addr := '1{10.13.50.77}3'); // SEN.ADDM
MY_WRITE_VAR(
    Execute := My_Addm.Done,
    Addr := My_Addr_Table,
    Timeout := 5,
    ObjType := SEN.ObjectType.MW,
    FirstObj := 68,
    Quantity := 4,
    Buffer := ADR(SEND_Buffer)); // WRITE_VAR
// My_Addr_Table: input not connected
// SEND_Buffer[0]: input not connected
// SEND_Buffer[1]: input not connected
// SEND_Buffer[2]: input not connected
// SEND_Buffer[3]: input not connected

END_PROGRAM

// DCCM_PCL_2/Application/LIBRARY/FB_PCMS_WATCHDOG
FUNCTION_BLOCK FB_PCMS_WATCHDOG
VAR_OUTPUT
	LAST_VALUE: INT;
END_VAR
VAR_INPUT
	VALUE: INT;
END_VAR
VAR_OUTPUT
	TIMEOUT: BOOL;
END_VAR
VAR
	START_DELAY_TON: TON;
END_VAR

START_DELAY_TON(IN := (LAST_VALUE = VALUE), PT := T#120S);
TIMEOUT := START_DELAY_TON.Q;

LAST_VALUE := VALUE;

END_FUNCTION_BLOCK
